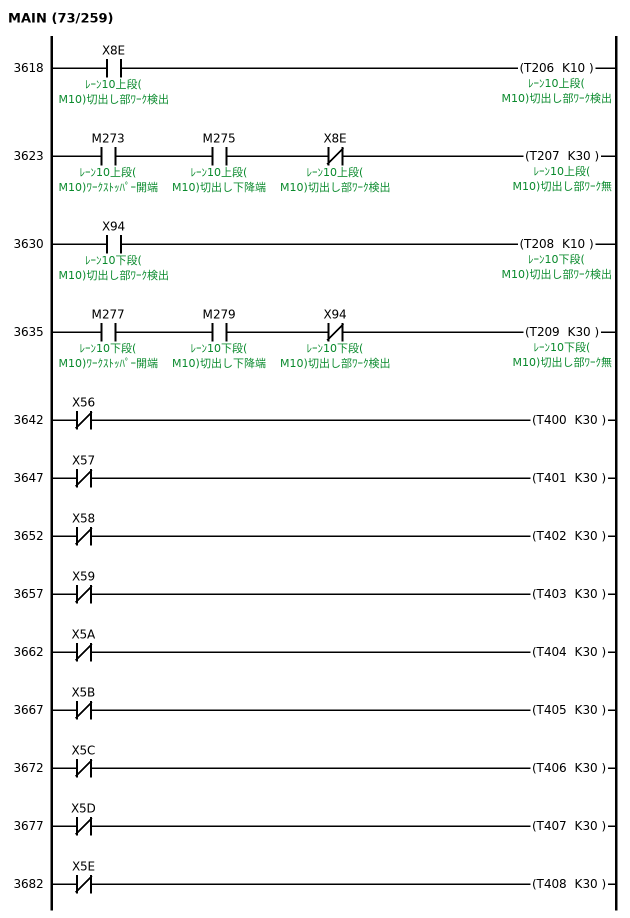
[picture p72: ladder of MAIN, rungs at steps 3618 to 3682]
3618  LD      X8E  ; ﾚｰﾝ10上段(M10)切出し部ﾜｰｸ検出
      OUT     T206 K10  ; ﾚｰﾝ10上段(M10)切出し部ﾜｰｸ検出
3623  LD      M273  ; ﾚｰﾝ10上段(M10)ﾜｰｸｽﾄｯﾊﾟｰ開端
      AND     M275  ; ﾚｰﾝ10上段(M10)切出し下降端
      ANI     X8E  ; ﾚｰﾝ10上段(M10)切出し部ﾜｰｸ検出
      OUT     T207 K30  ; ﾚｰﾝ10上段(M10)切出し部ﾜｰｸ無
3630  LD      X94  ; ﾚｰﾝ10下段(M10)切出し部ﾜｰｸ検出
      OUT     T208 K10  ; ﾚｰﾝ10下段(M10)切出し部ﾜｰｸ検出
3635  LD      M277  ; ﾚｰﾝ10下段(M10)ﾜｰｸｽﾄｯﾊﾟｰ開端
      AND     M279  ; ﾚｰﾝ10下段(M10)切出し下降端
      ANI     X94  ; ﾚｰﾝ10下段(M10)切出し部ﾜｰｸ検出
      OUT     T209 K30  ; ﾚｰﾝ10下段(M10)切出し部ﾜｰｸ無
3642  LDI     X56
      OUT     T400 K30
3647  LDI     X57
      OUT     T401 K30
3652  LDI     X58
      OUT     T402 K30
3657  LDI     X59
      OUT     T403 K30
3662  LDI     X5A
      OUT     T404 K30
3667  LDI     X5B
      OUT     T405 K30
3672  LDI     X5C
      OUT     T406 K30
3677  LDI     X5D
      OUT     T407 K30
3682  LDI     X5E
      OUT     T408 K30
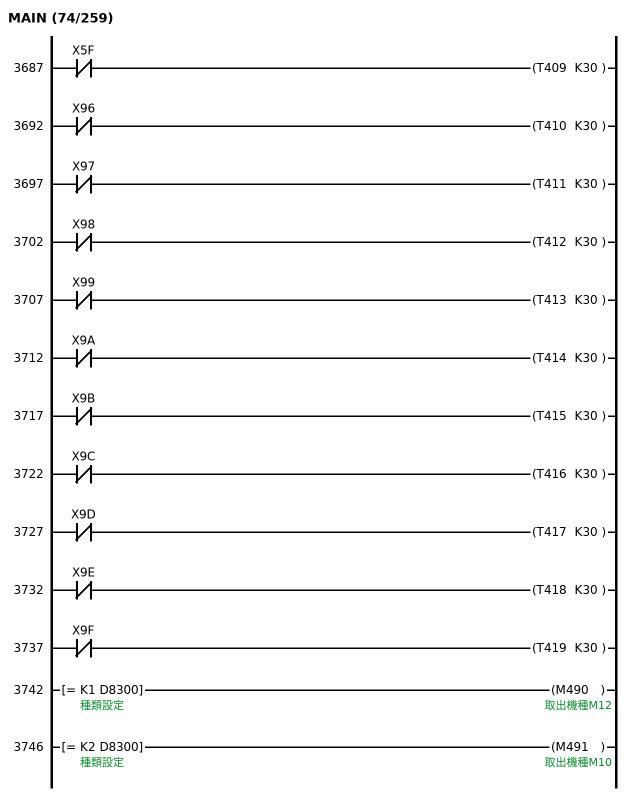
3687  LDI     X5F
      OUT     T409 K30
3692  LDI     X96
      OUT     T410 K30
3697  LDI     X97
      OUT     T411 K30
3702  LDI     X98
      OUT     T412 K30
3707  LDI     X99
      OUT     T413 K30
3712  LDI     X9A
      OUT     T414 K30
3717  LDI     X9B
      OUT     T415 K30
3722  LDI     X9C
      OUT     T416 K30
3727  LDI     X9D
      OUT     T417 K30
3732  LDI     X9E
      OUT     T418 K30
3737  LDI     X9F
      OUT     T419 K30
3742  LD=     K1 D8300  ; 種類設定
      OUT     M490  ; 取出機種M12
3746  LD=     K2 D8300  ; 種類設定
      OUT     M491  ; 取出機種M10
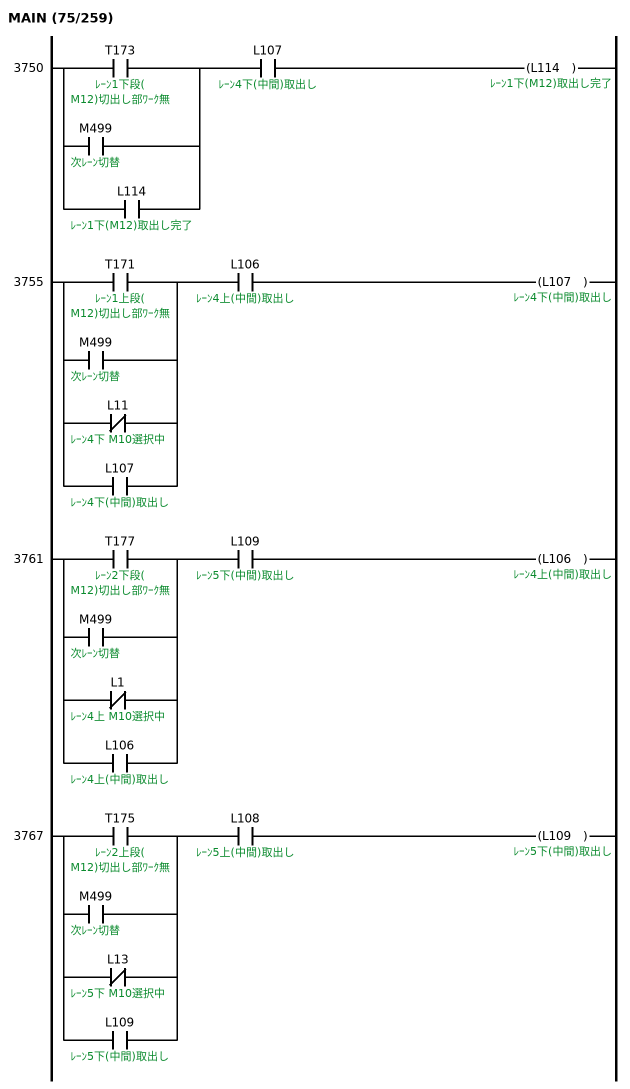
3750  LD      T173  ; ﾚｰﾝ1下段(M12)切出し部ﾜｰｸ無
      OR      M499  ; 次ﾚｰﾝ切替
      OR      L114  ; ﾚｰﾝ1下(M12)取出し完了
      AND     L107  ; ﾚｰﾝ4下(中間)取出し
      OUT     L114  ; ﾚｰﾝ1下(M12)取出し完了
3755  LD      T171  ; ﾚｰﾝ1上段(M12)切出し部ﾜｰｸ無
      OR      M499  ; 次ﾚｰﾝ切替
      ORI     L11  ; ﾚｰﾝ4下 M10選択中
      OR      L107  ; ﾚｰﾝ4下(中間)取出し
      AND     L106  ; ﾚｰﾝ4上(中間)取出し
      OUT     L107  ; ﾚｰﾝ4下(中間)取出し
3761  LD      T177  ; ﾚｰﾝ2下段(M12)切出し部ﾜｰｸ無
      OR      M499  ; 次ﾚｰﾝ切替
      ORI     L1  ; ﾚｰﾝ4上 M10選択中
      OR      L106  ; ﾚｰﾝ4上(中間)取出し
      AND     L109  ; ﾚｰﾝ5下(中間)取出し
      OUT     L106  ; ﾚｰﾝ4上(中間)取出し
3767  LD      T175  ; ﾚｰﾝ2上段(M12)切出し部ﾜｰｸ無
      OR      M499  ; 次ﾚｰﾝ切替
      ORI     L13  ; ﾚｰﾝ5下 M10選択中
      OR      L109  ; ﾚｰﾝ5下(中間)取出し
      AND     L108  ; ﾚｰﾝ5上(中間)取出し
      OUT     L109  ; ﾚｰﾝ5下(中間)取出し
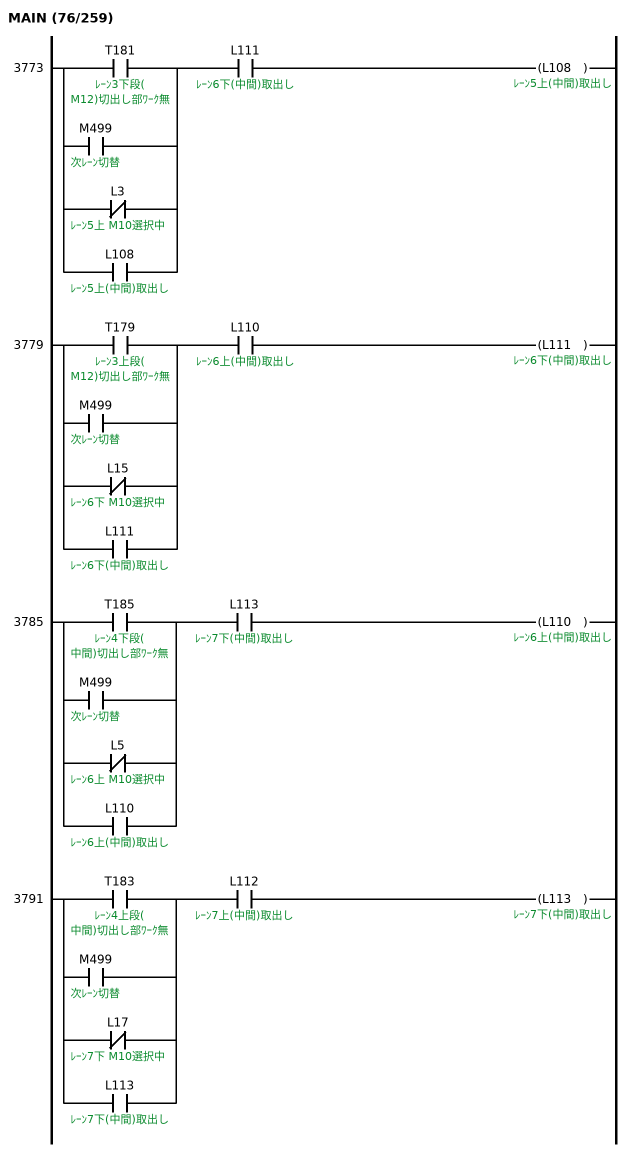
3773  LD      T181  ; ﾚｰﾝ3下段(M12)切出し部ﾜｰｸ無
      OR      M499  ; 次ﾚｰﾝ切替
      ORI     L3  ; ﾚｰﾝ5上 M10選択中
      OR      L108  ; ﾚｰﾝ5上(中間)取出し
      AND     L111  ; ﾚｰﾝ6下(中間)取出し
      OUT     L108  ; ﾚｰﾝ5上(中間)取出し
3779  LD      T179  ; ﾚｰﾝ3上段(M12)切出し部ﾜｰｸ無
      OR      M499  ; 次ﾚｰﾝ切替
      ORI     L15  ; ﾚｰﾝ6下 M10選択中
      OR      L111  ; ﾚｰﾝ6下(中間)取出し
      AND     L110  ; ﾚｰﾝ6上(中間)取出し
      OUT     L111  ; ﾚｰﾝ6下(中間)取出し
3785  LD      T185  ; ﾚｰﾝ4下段(中間)切出し部ﾜｰｸ無
      OR      M499  ; 次ﾚｰﾝ切替
      ORI     L5  ; ﾚｰﾝ6上 M10選択中
      OR      L110  ; ﾚｰﾝ6上(中間)取出し
      AND     L113  ; ﾚｰﾝ7下(中間)取出し
      OUT     L110  ; ﾚｰﾝ6上(中間)取出し
3791  LD      T183  ; ﾚｰﾝ4上段(中間)切出し部ﾜｰｸ無
      OR      M499  ; 次ﾚｰﾝ切替
      ORI     L17  ; ﾚｰﾝ7下 M10選択中
      OR      L113  ; ﾚｰﾝ7下(中間)取出し
      AND     L112  ; ﾚｰﾝ7上(中間)取出し
      OUT     L113  ; ﾚｰﾝ7下(中間)取出し
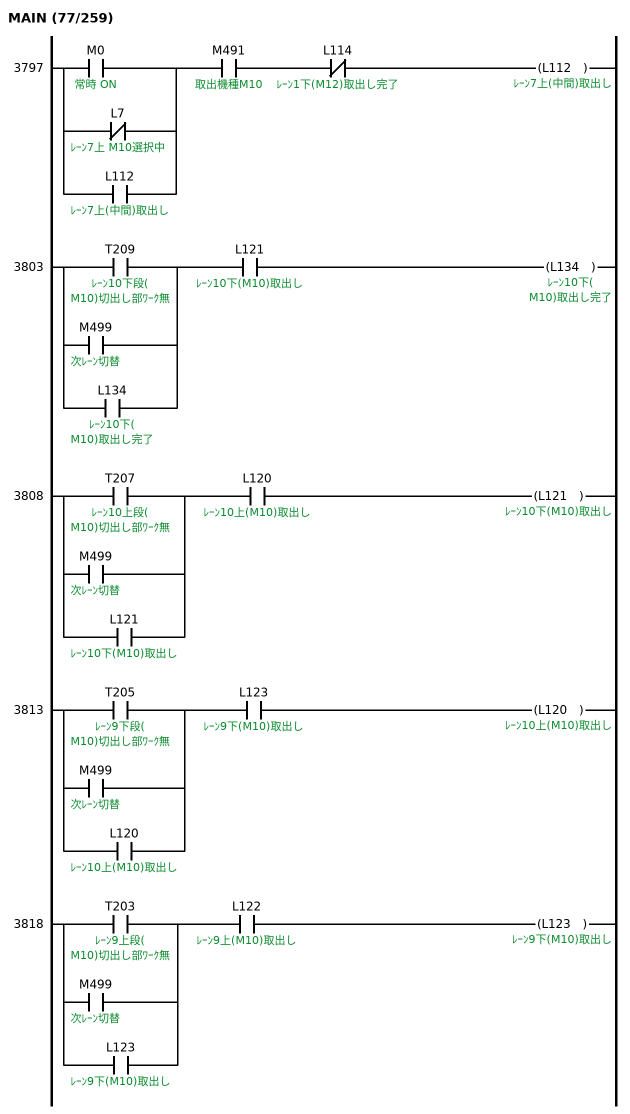
3797  LD      M0  ; 常時 ON
      ORI     L7  ; ﾚｰﾝ7上 M10選択中
      OR      L112  ; ﾚｰﾝ7上(中間)取出し
      AND     M491  ; 取出機種M10
      ANI     L114  ; ﾚｰﾝ1下(M12)取出し完了
      OUT     L112  ; ﾚｰﾝ7上(中間)取出し
3803  LD      T209  ; ﾚｰﾝ10下段(M10)切出し部ﾜｰｸ無
      OR      M499  ; 次ﾚｰﾝ切替
      OR      L134  ; ﾚｰﾝ10下(M10)取出し完了
      AND     L121  ; ﾚｰﾝ10下(M10)取出し
      OUT     L134  ; ﾚｰﾝ10下(M10)取出し完了
3808  LD      T207  ; ﾚｰﾝ10上段(M10)切出し部ﾜｰｸ無
      OR      M499  ; 次ﾚｰﾝ切替
      OR      L121  ; ﾚｰﾝ10下(M10)取出し
      AND     L120  ; ﾚｰﾝ10上(M10)取出し
      OUT     L121  ; ﾚｰﾝ10下(M10)取出し
3813  LD      T205  ; ﾚｰﾝ9下段(M10)切出し部ﾜｰｸ無
      OR      M499  ; 次ﾚｰﾝ切替
      OR      L120  ; ﾚｰﾝ10上(M10)取出し
      AND     L123  ; ﾚｰﾝ9下(M10)取出し
      OUT     L120  ; ﾚｰﾝ10上(M10)取出し
3818  LD      T203  ; ﾚｰﾝ9上段(M10)切出し部ﾜｰｸ無
      OR      M499  ; 次ﾚｰﾝ切替
      OR      L123  ; ﾚｰﾝ9下(M10)取出し
      AND     L122  ; ﾚｰﾝ9上(M10)取出し
      OUT     L123  ; ﾚｰﾝ9下(M10)取出し
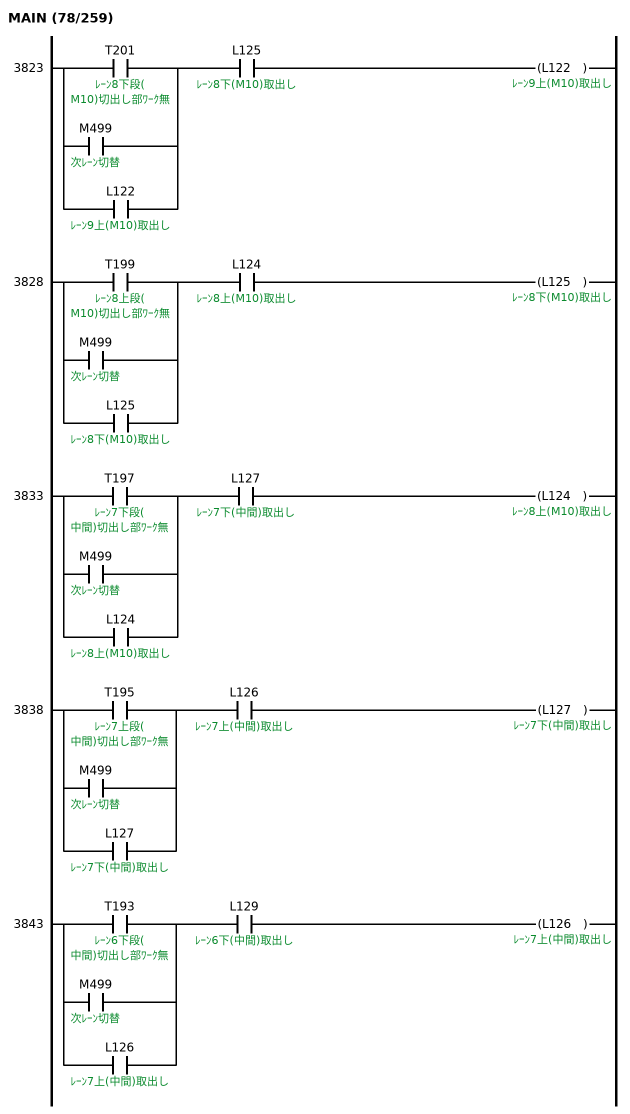
3823  LD      T201  ; ﾚｰﾝ8下段(M10)切出し部ﾜｰｸ無
      OR      M499  ; 次ﾚｰﾝ切替
      OR      L122  ; ﾚｰﾝ9上(M10)取出し
      AND     L125  ; ﾚｰﾝ8下(M10)取出し
      OUT     L122  ; ﾚｰﾝ9上(M10)取出し
3828  LD      T199  ; ﾚｰﾝ8上段(M10)切出し部ﾜｰｸ無
      OR      M499  ; 次ﾚｰﾝ切替
      OR      L125  ; ﾚｰﾝ8下(M10)取出し
      AND     L124  ; ﾚｰﾝ8上(M10)取出し
      OUT     L125  ; ﾚｰﾝ8下(M10)取出し
3833  LD      T197  ; ﾚｰﾝ7下段(中間)切出し部ﾜｰｸ無
      OR      M499  ; 次ﾚｰﾝ切替
      OR      L124  ; ﾚｰﾝ8上(M10)取出し
      AND     L127  ; ﾚｰﾝ7下(中間)取出し
      OUT     L124  ; ﾚｰﾝ8上(M10)取出し
3838  LD      T195  ; ﾚｰﾝ7上段(中間)切出し部ﾜｰｸ無
      OR      M499  ; 次ﾚｰﾝ切替
      OR      L127  ; ﾚｰﾝ7下(中間)取出し
      AND     L126  ; ﾚｰﾝ7上(中間)取出し
      OUT     L127  ; ﾚｰﾝ7下(中間)取出し
3843  LD      T193  ; ﾚｰﾝ6下段(中間)切出し部ﾜｰｸ無
      OR      M499  ; 次ﾚｰﾝ切替
      OR      L126  ; ﾚｰﾝ7上(中間)取出し
      AND     L129  ; ﾚｰﾝ6下(中間)取出し
      OUT     L126  ; ﾚｰﾝ7上(中間)取出し
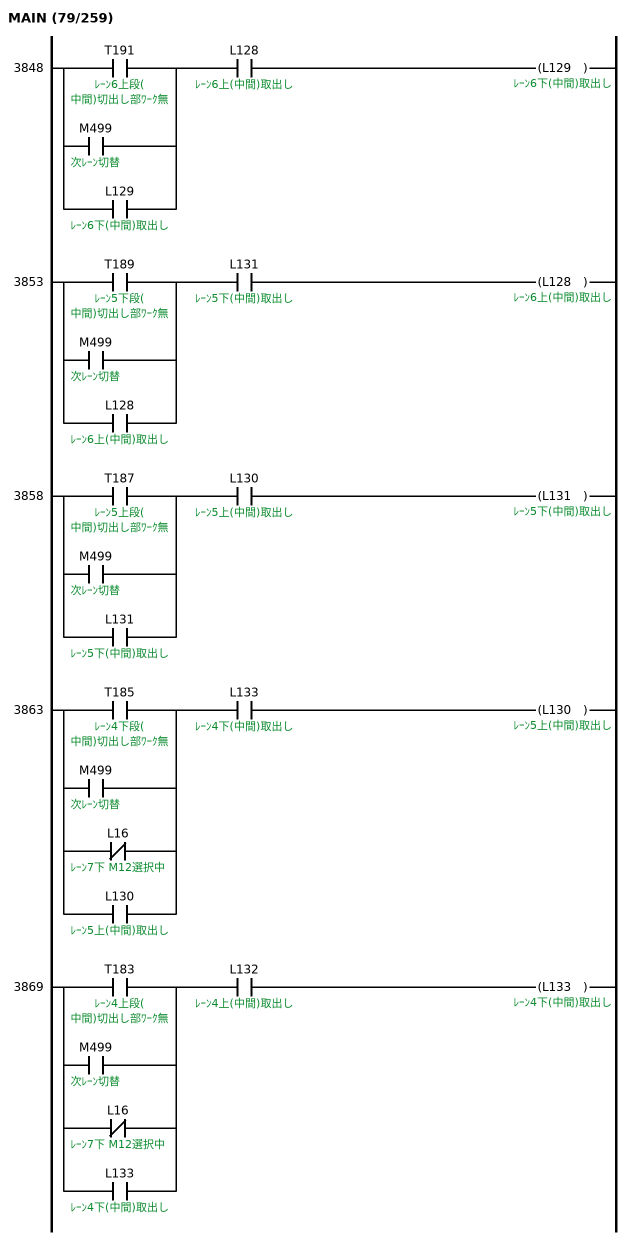
3848  LD      T191  ; ﾚｰﾝ6上段(中間)切出し部ﾜｰｸ無
      OR      M499  ; 次ﾚｰﾝ切替
      OR      L129  ; ﾚｰﾝ6下(中間)取出し
      AND     L128  ; ﾚｰﾝ6上(中間)取出し
      OUT     L129  ; ﾚｰﾝ6下(中間)取出し
3853  LD      T189  ; ﾚｰﾝ5下段(中間)切出し部ﾜｰｸ無
      OR      M499  ; 次ﾚｰﾝ切替
      OR      L128  ; ﾚｰﾝ6上(中間)取出し
      AND     L131  ; ﾚｰﾝ5下(中間)取出し
      OUT     L128  ; ﾚｰﾝ6上(中間)取出し
3858  LD      T187  ; ﾚｰﾝ5上段(中間)切出し部ﾜｰｸ無
      OR      M499  ; 次ﾚｰﾝ切替
      OR      L131  ; ﾚｰﾝ5下(中間)取出し
      AND     L130  ; ﾚｰﾝ5上(中間)取出し
      OUT     L131  ; ﾚｰﾝ5下(中間)取出し
3863  LD      T185  ; ﾚｰﾝ4下段(中間)切出し部ﾜｰｸ無
      OR      M499  ; 次ﾚｰﾝ切替
      ORI     L16  ; ﾚｰﾝ7下 M12選択中
      OR      L130  ; ﾚｰﾝ5上(中間)取出し
      AND     L133  ; ﾚｰﾝ4下(中間)取出し
      OUT     L130  ; ﾚｰﾝ5上(中間)取出し
3869  LD      T183  ; ﾚｰﾝ4上段(中間)切出し部ﾜｰｸ無
      OR      M499  ; 次ﾚｰﾝ切替
      ORI     L16  ; ﾚｰﾝ7下 M12選択中
      OR      L133  ; ﾚｰﾝ4下(中間)取出し
      AND     L132  ; ﾚｰﾝ4上(中間)取出し
      OUT     L133  ; ﾚｰﾝ4下(中間)取出し
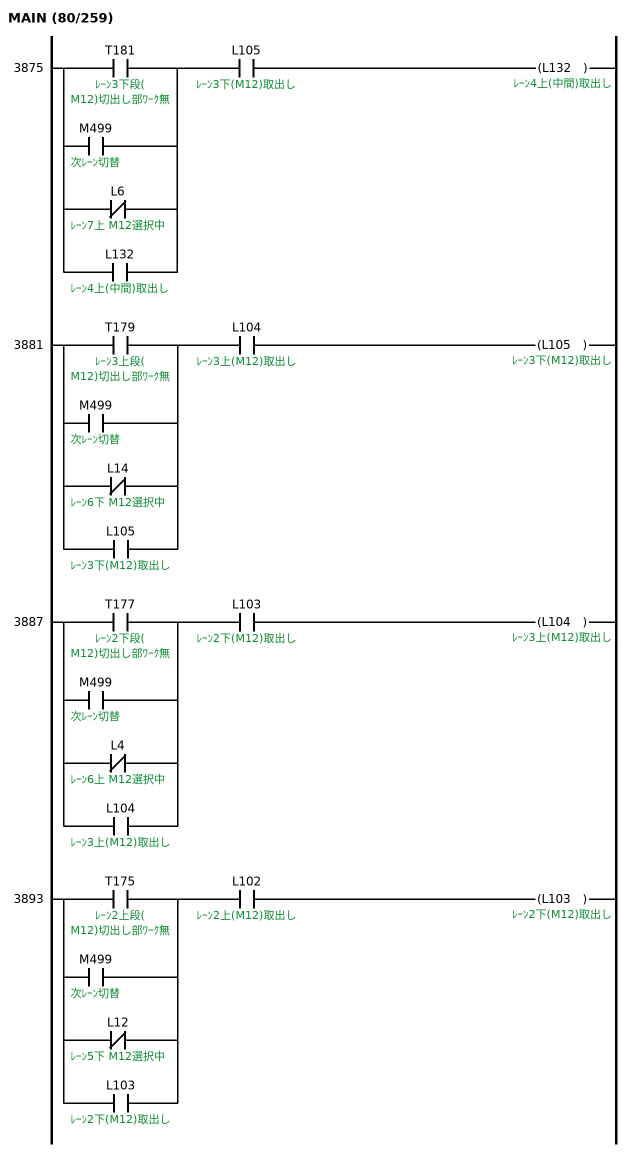
3875  LD      T181  ; ﾚｰﾝ3下段(M12)切出し部ﾜｰｸ無
      OR      M499  ; 次ﾚｰﾝ切替
      ORI     L6  ; ﾚｰﾝ7上 M12選択中
      OR      L132  ; ﾚｰﾝ4上(中間)取出し
      AND     L105  ; ﾚｰﾝ3下(M12)取出し
      OUT     L132  ; ﾚｰﾝ4上(中間)取出し
3881  LD      T179  ; ﾚｰﾝ3上段(M12)切出し部ﾜｰｸ無
      OR      M499  ; 次ﾚｰﾝ切替
      ORI     L14  ; ﾚｰﾝ6下 M12選択中
      OR      L105  ; ﾚｰﾝ3下(M12)取出し
      AND     L104  ; ﾚｰﾝ3上(M12)取出し
      OUT     L105  ; ﾚｰﾝ3下(M12)取出し
3887  LD      T177  ; ﾚｰﾝ2下段(M12)切出し部ﾜｰｸ無
      OR      M499  ; 次ﾚｰﾝ切替
      ORI     L4  ; ﾚｰﾝ6上 M12選択中
      OR      L104  ; ﾚｰﾝ3上(M12)取出し
      AND     L103  ; ﾚｰﾝ2下(M12)取出し
      OUT     L104  ; ﾚｰﾝ3上(M12)取出し
3893  LD      T175  ; ﾚｰﾝ2上段(M12)切出し部ﾜｰｸ無
      OR      M499  ; 次ﾚｰﾝ切替
      ORI     L12  ; ﾚｰﾝ5下 M12選択中
      OR      L103  ; ﾚｰﾝ2下(M12)取出し
      AND     L102  ; ﾚｰﾝ2上(M12)取出し
      OUT     L103  ; ﾚｰﾝ2下(M12)取出し
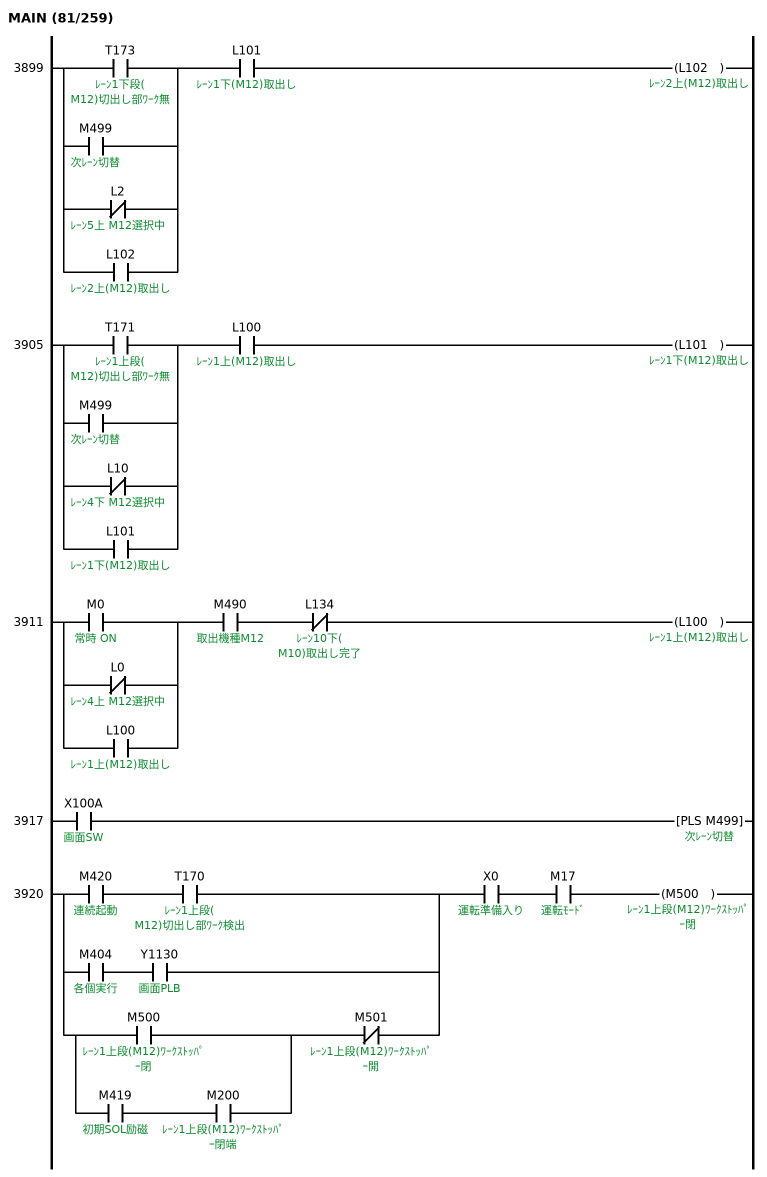
3899  LD      T173  ; ﾚｰﾝ1下段(M12)切出し部ﾜｰｸ無
      OR      M499  ; 次ﾚｰﾝ切替
      ORI     L2  ; ﾚｰﾝ5上 M12選択中
      OR      L102  ; ﾚｰﾝ2上(M12)取出し
      AND     L101  ; ﾚｰﾝ1下(M12)取出し
      OUT     L102  ; ﾚｰﾝ2上(M12)取出し
3905  LD      T171  ; ﾚｰﾝ1上段(M12)切出し部ﾜｰｸ無
      OR      M499  ; 次ﾚｰﾝ切替
      ORI     L10  ; ﾚｰﾝ4下 M12選択中
      OR      L101  ; ﾚｰﾝ1下(M12)取出し
      AND     L100  ; ﾚｰﾝ1上(M12)取出し
      OUT     L101  ; ﾚｰﾝ1下(M12)取出し
3911  LD      M0  ; 常時 ON
      ORI     L0  ; ﾚｰﾝ4上 M12選択中
      OR      L100  ; ﾚｰﾝ1上(M12)取出し
      AND     M490  ; 取出機種M12
      ANI     L134  ; ﾚｰﾝ10下(M10)取出し完了
      OUT     L100  ; ﾚｰﾝ1上(M12)取出し
3917  LD      X100A  ; 画面SW
      PLS     M499  ; 次ﾚｰﾝ切替
3920  LD      M420  ; 連続起動
      AND     T170  ; ﾚｰﾝ1上段(M12)切出し部ﾜｰｸ検出
      LD      M404  ; 各個実行
      AND     Y1130  ; 画面PLB
      ORB
      LD      M500  ; ﾚｰﾝ1上段(M12)ﾜｰｸｽﾄｯﾊﾟｰ閉
      LD      M419  ; 初期SOL励磁
      AND     M200  ; ﾚｰﾝ1上段(M12)ﾜｰｸｽﾄｯﾊﾟｰ閉端
      ORB
      ANI     M501  ; ﾚｰﾝ1上段(M12)ﾜｰｸｽﾄｯﾊﾟｰ開
      ORB
      AND     X0  ; 運転準備入り
      AND     M17  ; 運転ﾓｰﾄﾞ
      OUT     M500  ; ﾚｰﾝ1上段(M12)ﾜｰｸｽﾄｯﾊﾟｰ閉
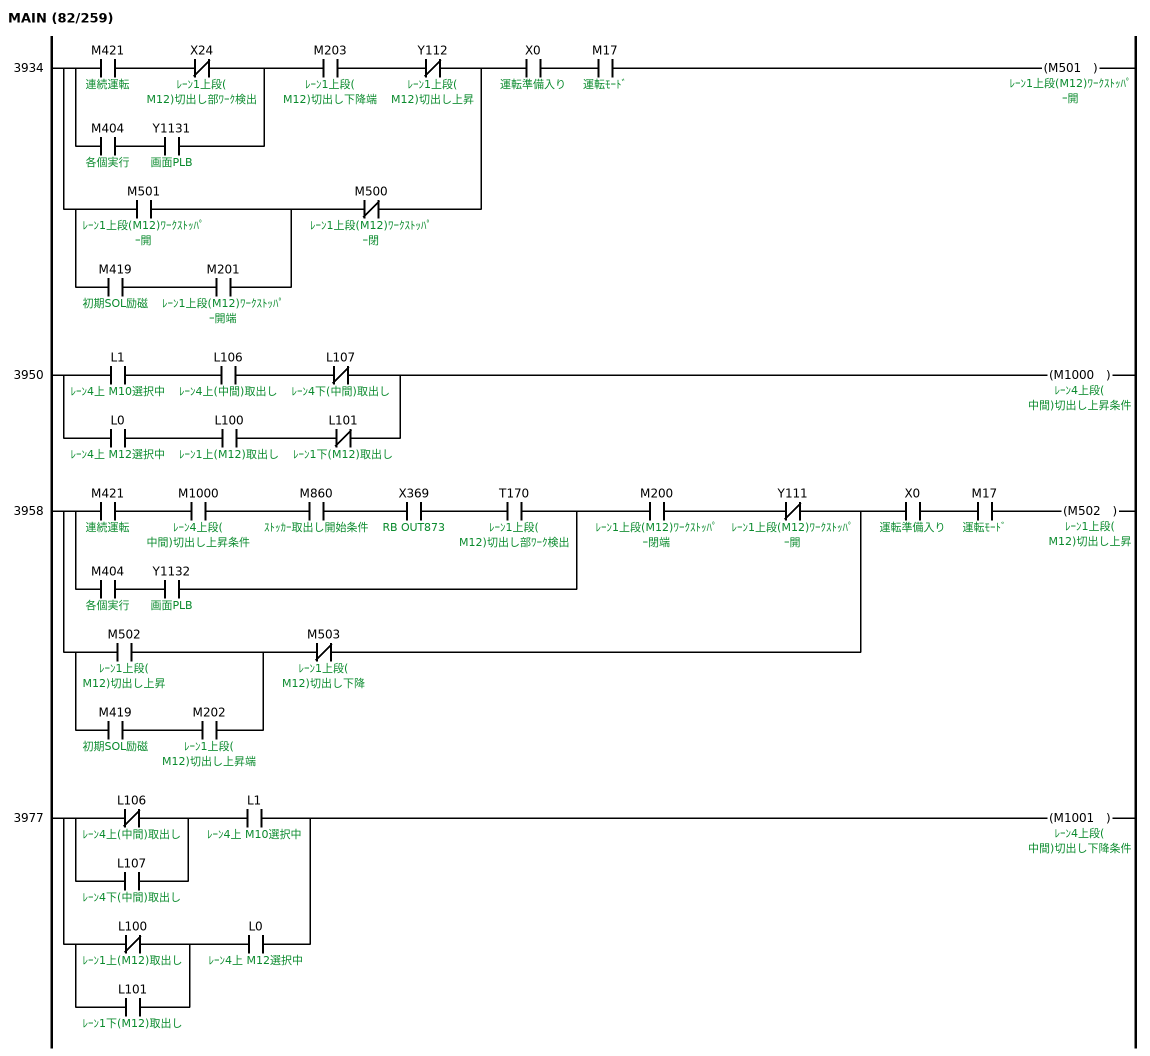
3934  LD      M421  ; 連続運転
      ANI     X24  ; ﾚｰﾝ1上段(M12)切出し部ﾜｰｸ検出
      LD      M404  ; 各個実行
      AND     Y1131  ; 画面PLB
      ORB
      AND     M203  ; ﾚｰﾝ1上段(M12)切出し下降端
      ANI     Y112  ; ﾚｰﾝ1上段(M12)切出し上昇
      LD      M501  ; ﾚｰﾝ1上段(M12)ﾜｰｸｽﾄｯﾊﾟｰ開
      LD      M419  ; 初期SOL励磁
      AND     M201  ; ﾚｰﾝ1上段(M12)ﾜｰｸｽﾄｯﾊﾟｰ開端
      ORB
      ANI     M500  ; ﾚｰﾝ1上段(M12)ﾜｰｸｽﾄｯﾊﾟｰ閉
      ORB
      AND     X0  ; 運転準備入り
      AND     M17  ; 運転ﾓｰﾄﾞ
      OUT     M501  ; ﾚｰﾝ1上段(M12)ﾜｰｸｽﾄｯﾊﾟｰ開
3950  LD      L1  ; ﾚｰﾝ4上 M10選択中
      AND     L106  ; ﾚｰﾝ4上(中間)取出し
      ANI     L107  ; ﾚｰﾝ4下(中間)取出し
      LD      L0  ; ﾚｰﾝ4上 M12選択中
      AND     L100  ; ﾚｰﾝ1上(M12)取出し
      ANI     L101  ; ﾚｰﾝ1下(M12)取出し
      ORB
      OUT     M1000  ; ﾚｰﾝ4上段(中間)切出し上昇条件
3958  LD      M421  ; 連続運転
      AND     M1000  ; ﾚｰﾝ4上段(中間)切出し上昇条件
      AND     M860  ; ｽﾄｯｶｰ取出し開始条件
      AND     X369  ; RB OUT873
      AND     T170  ; ﾚｰﾝ1上段(M12)切出し部ﾜｰｸ検出
      LD      M404  ; 各個実行
      AND     Y1132  ; 画面PLB
      ORB
      AND     M200  ; ﾚｰﾝ1上段(M12)ﾜｰｸｽﾄｯﾊﾟｰ閉端
      ANI     Y111  ; ﾚｰﾝ1上段(M12)ﾜｰｸｽﾄｯﾊﾟｰ開
      LD      M502  ; ﾚｰﾝ1上段(M12)切出し上昇
      LD      M419  ; 初期SOL励磁
      AND     M202  ; ﾚｰﾝ1上段(M12)切出し上昇端
      ORB
      ANI     M503  ; ﾚｰﾝ1上段(M12)切出し下降
      ORB
      AND     X0  ; 運転準備入り
      AND     M17  ; 運転ﾓｰﾄﾞ
      OUT     M502  ; ﾚｰﾝ1上段(M12)切出し上昇
3977  LDI     L106  ; ﾚｰﾝ4上(中間)取出し
      OR      L107  ; ﾚｰﾝ4下(中間)取出し
      AND     L1  ; ﾚｰﾝ4上 M10選択中
      LDI     L100  ; ﾚｰﾝ1上(M12)取出し
      OR      L101  ; ﾚｰﾝ1下(M12)取出し
      AND     L0  ; ﾚｰﾝ4上 M12選択中
      ORB
      OUT     M1001  ; ﾚｰﾝ4上段(中間)切出し下降条件
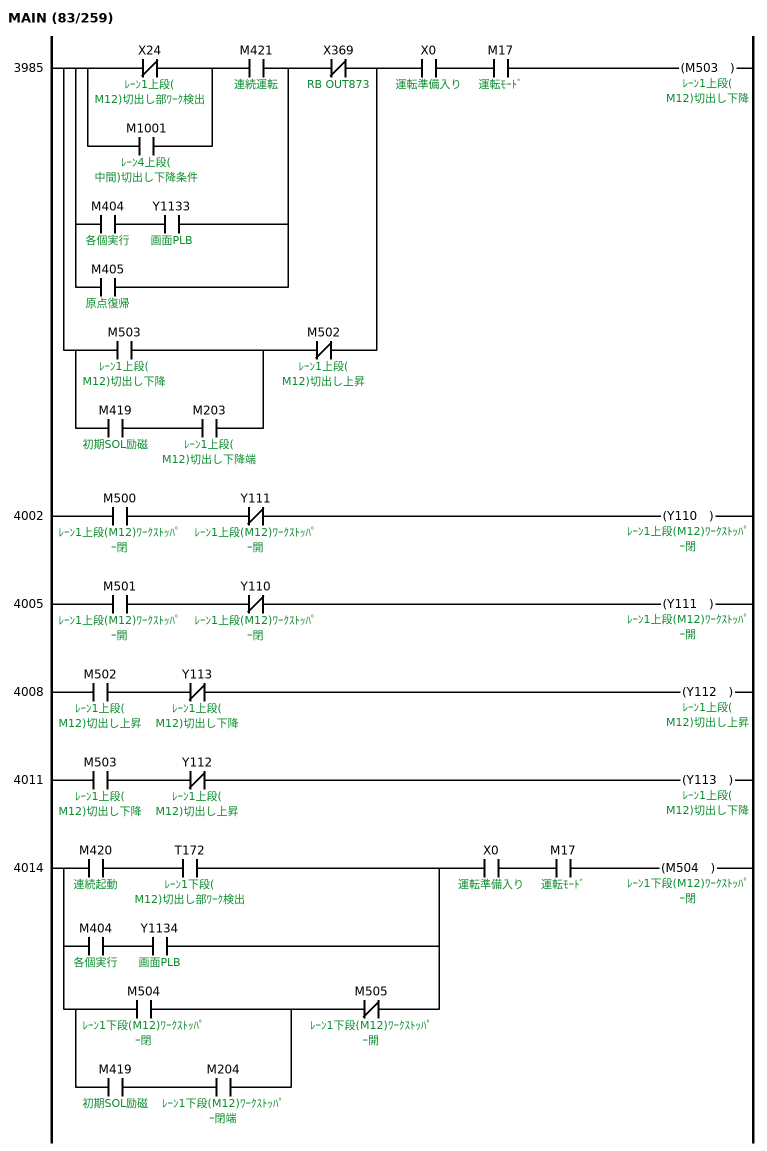
3985  LDI     X24  ; ﾚｰﾝ1上段(M12)切出し部ﾜｰｸ検出
      OR      M1001  ; ﾚｰﾝ4上段(中間)切出し下降条件
      AND     M421  ; 連続運転
      LD      M404  ; 各個実行
      AND     Y1133  ; 画面PLB
      ORB
      OR      M405  ; 原点復帰
      ANI     X369  ; RB OUT873
      LD      M503  ; ﾚｰﾝ1上段(M12)切出し下降
      LD      M419  ; 初期SOL励磁
      AND     M203  ; ﾚｰﾝ1上段(M12)切出し下降端
      ORB
      ANI     M502  ; ﾚｰﾝ1上段(M12)切出し上昇
      ORB
      AND     X0  ; 運転準備入り
      AND     M17  ; 運転ﾓｰﾄﾞ
      OUT     M503  ; ﾚｰﾝ1上段(M12)切出し下降
4002  LD      M500  ; ﾚｰﾝ1上段(M12)ﾜｰｸｽﾄｯﾊﾟｰ閉
      ANI     Y111  ; ﾚｰﾝ1上段(M12)ﾜｰｸｽﾄｯﾊﾟｰ開
      OUT     Y110  ; ﾚｰﾝ1上段(M12)ﾜｰｸｽﾄｯﾊﾟｰ閉
4005  LD      M501  ; ﾚｰﾝ1上段(M12)ﾜｰｸｽﾄｯﾊﾟｰ開
      ANI     Y110  ; ﾚｰﾝ1上段(M12)ﾜｰｸｽﾄｯﾊﾟｰ閉
      OUT     Y111  ; ﾚｰﾝ1上段(M12)ﾜｰｸｽﾄｯﾊﾟｰ開
4008  LD      M502  ; ﾚｰﾝ1上段(M12)切出し上昇
      ANI     Y113  ; ﾚｰﾝ1上段(M12)切出し下降
      OUT     Y112  ; ﾚｰﾝ1上段(M12)切出し上昇
4011  LD      M503  ; ﾚｰﾝ1上段(M12)切出し下降
      ANI     Y112  ; ﾚｰﾝ1上段(M12)切出し上昇
      OUT     Y113  ; ﾚｰﾝ1上段(M12)切出し下降
4014  LD      M420  ; 連続起動
      AND     T172  ; ﾚｰﾝ1下段(M12)切出し部ﾜｰｸ検出
      LD      M404  ; 各個実行
      AND     Y1134  ; 画面PLB
      ORB
      LD      M504  ; ﾚｰﾝ1下段(M12)ﾜｰｸｽﾄｯﾊﾟｰ閉
      LD      M419  ; 初期SOL励磁
      AND     M204  ; ﾚｰﾝ1下段(M12)ﾜｰｸｽﾄｯﾊﾟｰ閉端
      ORB
      ANI     M505  ; ﾚｰﾝ1下段(M12)ﾜｰｸｽﾄｯﾊﾟｰ開
      ORB
      AND     X0  ; 運転準備入り
      AND     M17  ; 運転ﾓｰﾄﾞ
      OUT     M504  ; ﾚｰﾝ1下段(M12)ﾜｰｸｽﾄｯﾊﾟｰ閉
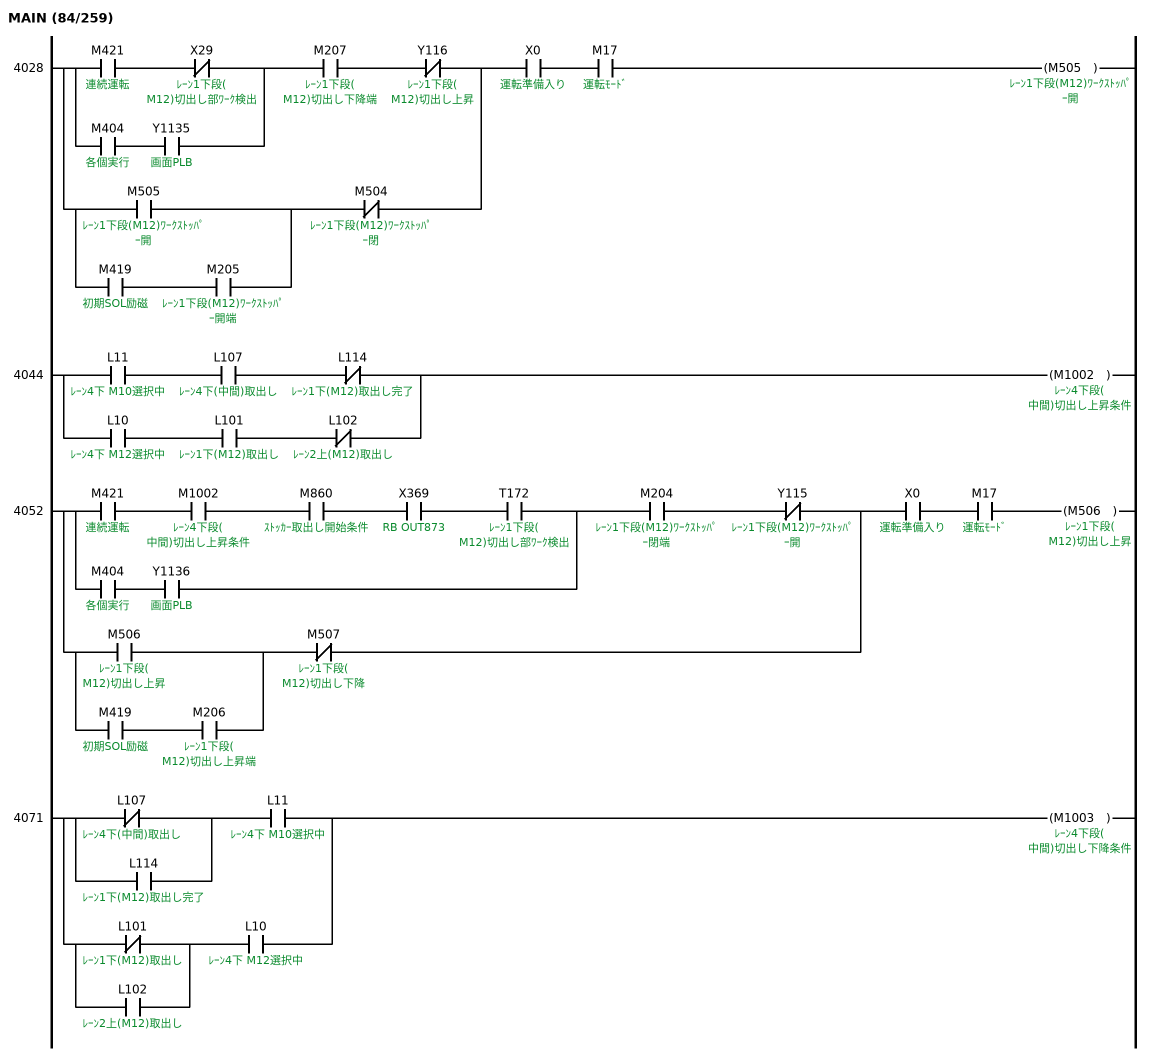
4028  LD      M421  ; 連続運転
      ANI     X29  ; ﾚｰﾝ1下段(M12)切出し部ﾜｰｸ検出
      LD      M404  ; 各個実行
      AND     Y1135  ; 画面PLB
      ORB
      AND     M207  ; ﾚｰﾝ1下段(M12)切出し下降端
      ANI     Y116  ; ﾚｰﾝ1下段(M12)切出し上昇
      LD      M505  ; ﾚｰﾝ1下段(M12)ﾜｰｸｽﾄｯﾊﾟｰ開
      LD      M419  ; 初期SOL励磁
      AND     M205  ; ﾚｰﾝ1下段(M12)ﾜｰｸｽﾄｯﾊﾟｰ開端
      ORB
      ANI     M504  ; ﾚｰﾝ1下段(M12)ﾜｰｸｽﾄｯﾊﾟｰ閉
      ORB
      AND     X0  ; 運転準備入り
      AND     M17  ; 運転ﾓｰﾄﾞ
      OUT     M505  ; ﾚｰﾝ1下段(M12)ﾜｰｸｽﾄｯﾊﾟｰ開
4044  LD      L11  ; ﾚｰﾝ4下 M10選択中
      AND     L107  ; ﾚｰﾝ4下(中間)取出し
      ANI     L114  ; ﾚｰﾝ1下(M12)取出し完了
      LD      L10  ; ﾚｰﾝ4下 M12選択中
      AND     L101  ; ﾚｰﾝ1下(M12)取出し
      ANI     L102  ; ﾚｰﾝ2上(M12)取出し
      ORB
      OUT     M1002  ; ﾚｰﾝ4下段(中間)切出し上昇条件
4052  LD      M421  ; 連続運転
      AND     M1002  ; ﾚｰﾝ4下段(中間)切出し上昇条件
      AND     M860  ; ｽﾄｯｶｰ取出し開始条件
      AND     X369  ; RB OUT873
      AND     T172  ; ﾚｰﾝ1下段(M12)切出し部ﾜｰｸ検出
      LD      M404  ; 各個実行
      AND     Y1136  ; 画面PLB
      ORB
      AND     M204  ; ﾚｰﾝ1下段(M12)ﾜｰｸｽﾄｯﾊﾟｰ閉端
      ANI     Y115  ; ﾚｰﾝ1下段(M12)ﾜｰｸｽﾄｯﾊﾟｰ開
      LD      M506  ; ﾚｰﾝ1下段(M12)切出し上昇
      LD      M419  ; 初期SOL励磁
      AND     M206  ; ﾚｰﾝ1下段(M12)切出し上昇端
      ORB
      ANI     M507  ; ﾚｰﾝ1下段(M12)切出し下降
      ORB
      AND     X0  ; 運転準備入り
      AND     M17  ; 運転ﾓｰﾄﾞ
      OUT     M506  ; ﾚｰﾝ1下段(M12)切出し上昇
4071  LDI     L107  ; ﾚｰﾝ4下(中間)取出し
      OR      L114  ; ﾚｰﾝ1下(M12)取出し完了
      AND     L11  ; ﾚｰﾝ4下 M10選択中
      LDI     L101  ; ﾚｰﾝ1下(M12)取出し
      OR      L102  ; ﾚｰﾝ2上(M12)取出し
      AND     L10  ; ﾚｰﾝ4下 M12選択中
      ORB
      OUT     M1003  ; ﾚｰﾝ4下段(中間)切出し下降条件
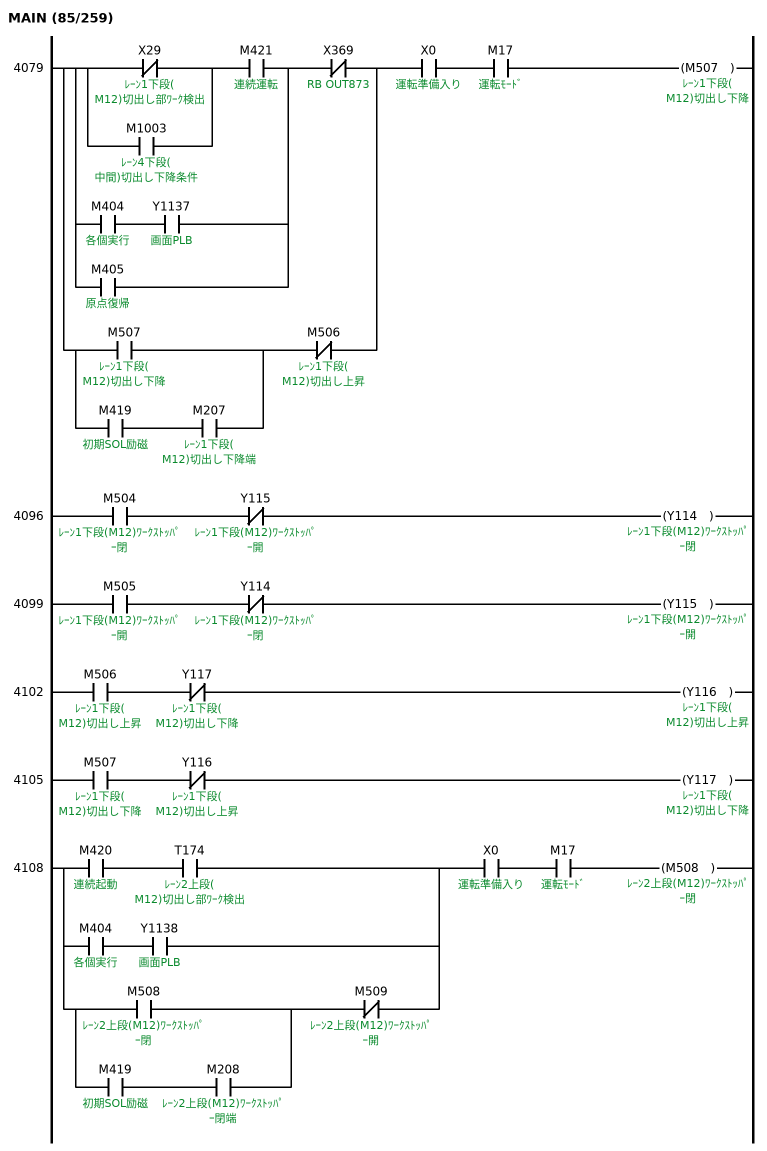
4079  LDI     X29  ; ﾚｰﾝ1下段(M12)切出し部ﾜｰｸ検出
      OR      M1003  ; ﾚｰﾝ4下段(中間)切出し下降条件
      AND     M421  ; 連続運転
      LD      M404  ; 各個実行
      AND     Y1137  ; 画面PLB
      ORB
      OR      M405  ; 原点復帰
      ANI     X369  ; RB OUT873
      LD      M507  ; ﾚｰﾝ1下段(M12)切出し下降
      LD      M419  ; 初期SOL励磁
      AND     M207  ; ﾚｰﾝ1下段(M12)切出し下降端
      ORB
      ANI     M506  ; ﾚｰﾝ1下段(M12)切出し上昇
      ORB
      AND     X0  ; 運転準備入り
      AND     M17  ; 運転ﾓｰﾄﾞ
      OUT     M507  ; ﾚｰﾝ1下段(M12)切出し下降
4096  LD      M504  ; ﾚｰﾝ1下段(M12)ﾜｰｸｽﾄｯﾊﾟｰ閉
      ANI     Y115  ; ﾚｰﾝ1下段(M12)ﾜｰｸｽﾄｯﾊﾟｰ開
      OUT     Y114  ; ﾚｰﾝ1下段(M12)ﾜｰｸｽﾄｯﾊﾟｰ閉
4099  LD      M505  ; ﾚｰﾝ1下段(M12)ﾜｰｸｽﾄｯﾊﾟｰ開
      ANI     Y114  ; ﾚｰﾝ1下段(M12)ﾜｰｸｽﾄｯﾊﾟｰ閉
      OUT     Y115  ; ﾚｰﾝ1下段(M12)ﾜｰｸｽﾄｯﾊﾟｰ開
4102  LD      M506  ; ﾚｰﾝ1下段(M12)切出し上昇
      ANI     Y117  ; ﾚｰﾝ1下段(M12)切出し下降
      OUT     Y116  ; ﾚｰﾝ1下段(M12)切出し上昇
4105  LD      M507  ; ﾚｰﾝ1下段(M12)切出し下降
      ANI     Y116  ; ﾚｰﾝ1下段(M12)切出し上昇
      OUT     Y117  ; ﾚｰﾝ1下段(M12)切出し下降
4108  LD      M420  ; 連続起動
      AND     T174  ; ﾚｰﾝ2上段(M12)切出し部ﾜｰｸ検出
      LD      M404  ; 各個実行
      AND     Y1138  ; 画面PLB
      ORB
      LD      M508  ; ﾚｰﾝ2上段(M12)ﾜｰｸｽﾄｯﾊﾟｰ閉
      LD      M419  ; 初期SOL励磁
      AND     M208  ; ﾚｰﾝ2上段(M12)ﾜｰｸｽﾄｯﾊﾟｰ閉端
      ORB
      ANI     M509  ; ﾚｰﾝ2上段(M12)ﾜｰｸｽﾄｯﾊﾟｰ開
      ORB
      AND     X0  ; 運転準備入り
      AND     M17  ; 運転ﾓｰﾄﾞ
      OUT     M508  ; ﾚｰﾝ2上段(M12)ﾜｰｸｽﾄｯﾊﾟｰ閉
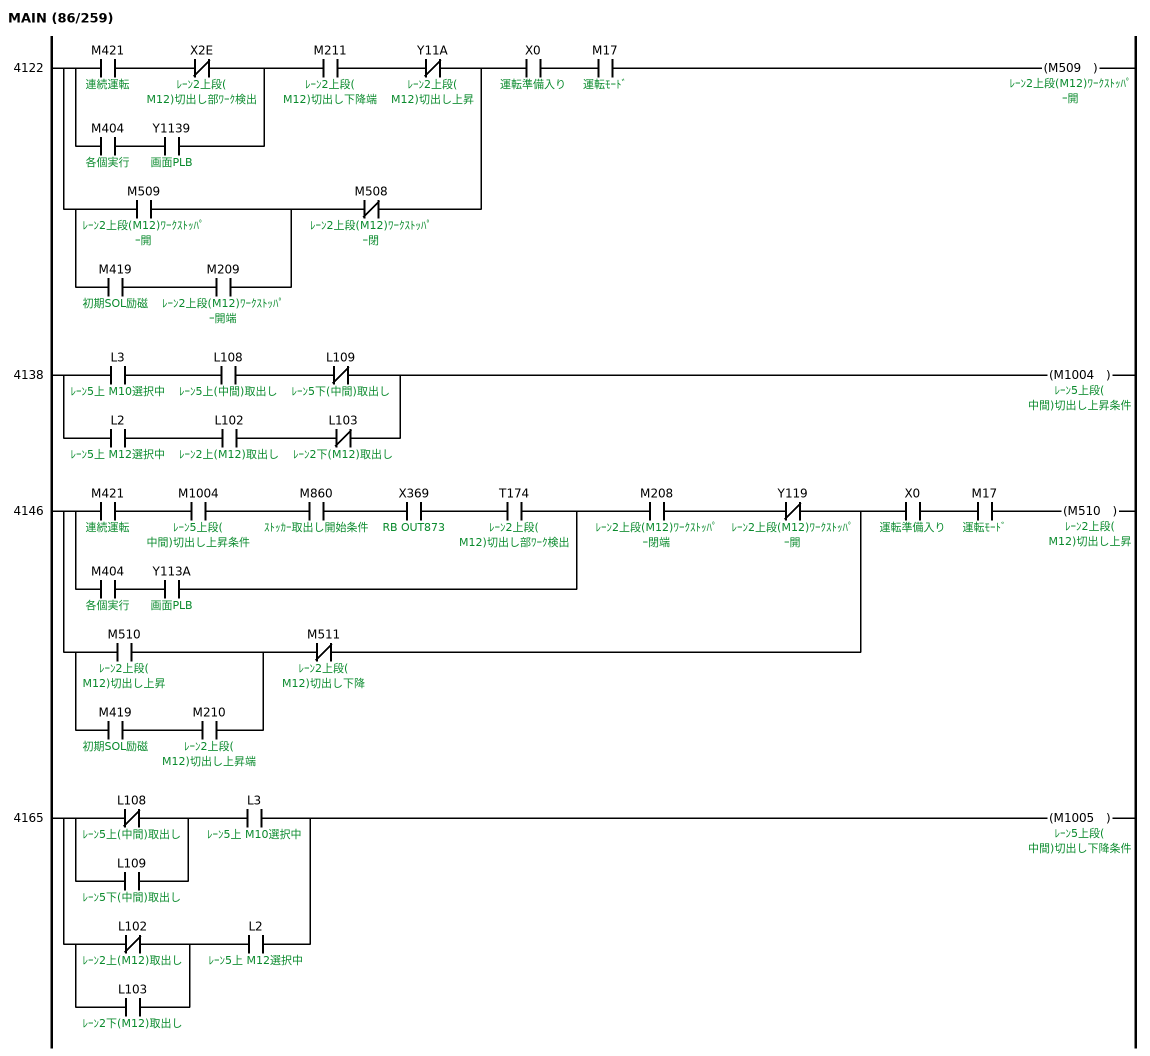
4122  LD      M421  ; 連続運転
      ANI     X2E  ; ﾚｰﾝ2上段(M12)切出し部ﾜｰｸ検出
      LD      M404  ; 各個実行
      AND     Y1139  ; 画面PLB
      ORB
      AND     M211  ; ﾚｰﾝ2上段(M12)切出し下降端
      ANI     Y11A  ; ﾚｰﾝ2上段(M12)切出し上昇
      LD      M509  ; ﾚｰﾝ2上段(M12)ﾜｰｸｽﾄｯﾊﾟｰ開
      LD      M419  ; 初期SOL励磁
      AND     M209  ; ﾚｰﾝ2上段(M12)ﾜｰｸｽﾄｯﾊﾟｰ開端
      ORB
      ANI     M508  ; ﾚｰﾝ2上段(M12)ﾜｰｸｽﾄｯﾊﾟｰ閉
      ORB
      AND     X0  ; 運転準備入り
      AND     M17  ; 運転ﾓｰﾄﾞ
      OUT     M509  ; ﾚｰﾝ2上段(M12)ﾜｰｸｽﾄｯﾊﾟｰ開
4138  LD      L3  ; ﾚｰﾝ5上 M10選択中
      AND     L108  ; ﾚｰﾝ5上(中間)取出し
      ANI     L109  ; ﾚｰﾝ5下(中間)取出し
      LD      L2  ; ﾚｰﾝ5上 M12選択中
      AND     L102  ; ﾚｰﾝ2上(M12)取出し
      ANI     L103  ; ﾚｰﾝ2下(M12)取出し
      ORB
      OUT     M1004  ; ﾚｰﾝ5上段(中間)切出し上昇条件
4146  LD      M421  ; 連続運転
      AND     M1004  ; ﾚｰﾝ5上段(中間)切出し上昇条件
      AND     M860  ; ｽﾄｯｶｰ取出し開始条件
      AND     X369  ; RB OUT873
      AND     T174  ; ﾚｰﾝ2上段(M12)切出し部ﾜｰｸ検出
      LD      M404  ; 各個実行
      AND     Y113A  ; 画面PLB
      ORB
      AND     M208  ; ﾚｰﾝ2上段(M12)ﾜｰｸｽﾄｯﾊﾟｰ閉端
      ANI     Y119  ; ﾚｰﾝ2上段(M12)ﾜｰｸｽﾄｯﾊﾟｰ開
      LD      M510  ; ﾚｰﾝ2上段(M12)切出し上昇
      LD      M419  ; 初期SOL励磁
      AND     M210  ; ﾚｰﾝ2上段(M12)切出し上昇端
      ORB
      ANI     M511  ; ﾚｰﾝ2上段(M12)切出し下降
      ORB
      AND     X0  ; 運転準備入り
      AND     M17  ; 運転ﾓｰﾄﾞ
      OUT     M510  ; ﾚｰﾝ2上段(M12)切出し上昇
4165  LDI     L108  ; ﾚｰﾝ5上(中間)取出し
      OR      L109  ; ﾚｰﾝ5下(中間)取出し
      AND     L3  ; ﾚｰﾝ5上 M10選択中
      LDI     L102  ; ﾚｰﾝ2上(M12)取出し
      OR      L103  ; ﾚｰﾝ2下(M12)取出し
      AND     L2  ; ﾚｰﾝ5上 M12選択中
      ORB
      OUT     M1005  ; ﾚｰﾝ5上段(中間)切出し下降条件
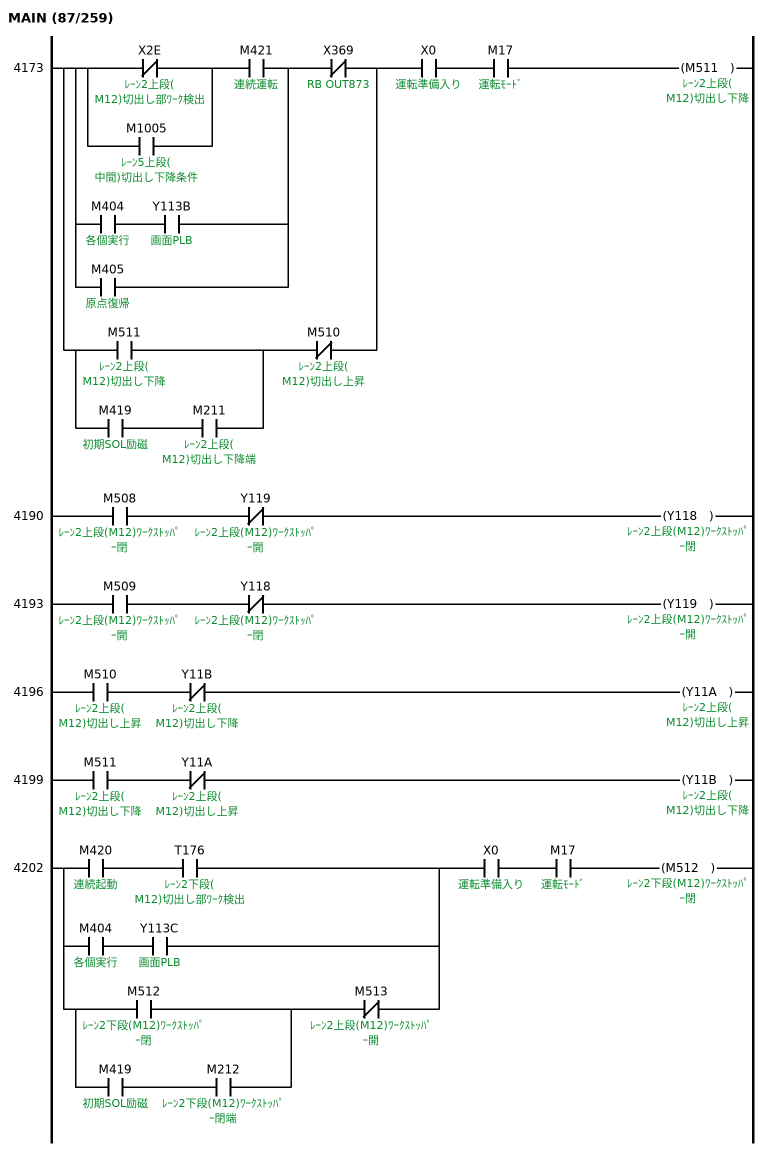
4173  LDI     X2E  ; ﾚｰﾝ2上段(M12)切出し部ﾜｰｸ検出
      OR      M1005  ; ﾚｰﾝ5上段(中間)切出し下降条件
      AND     M421  ; 連続運転
      LD      M404  ; 各個実行
      AND     Y113B  ; 画面PLB
      ORB
      OR      M405  ; 原点復帰
      ANI     X369  ; RB OUT873
      LD      M511  ; ﾚｰﾝ2上段(M12)切出し下降
      LD      M419  ; 初期SOL励磁
      AND     M211  ; ﾚｰﾝ2上段(M12)切出し下降端
      ORB
      ANI     M510  ; ﾚｰﾝ2上段(M12)切出し上昇
      ORB
      AND     X0  ; 運転準備入り
      AND     M17  ; 運転ﾓｰﾄﾞ
      OUT     M511  ; ﾚｰﾝ2上段(M12)切出し下降
4190  LD      M508  ; ﾚｰﾝ2上段(M12)ﾜｰｸｽﾄｯﾊﾟｰ閉
      ANI     Y119  ; ﾚｰﾝ2上段(M12)ﾜｰｸｽﾄｯﾊﾟｰ開
      OUT     Y118  ; ﾚｰﾝ2上段(M12)ﾜｰｸｽﾄｯﾊﾟｰ閉
4193  LD      M509  ; ﾚｰﾝ2上段(M12)ﾜｰｸｽﾄｯﾊﾟｰ開
      ANI     Y118  ; ﾚｰﾝ2上段(M12)ﾜｰｸｽﾄｯﾊﾟｰ閉
      OUT     Y119  ; ﾚｰﾝ2上段(M12)ﾜｰｸｽﾄｯﾊﾟｰ開
4196  LD      M510  ; ﾚｰﾝ2上段(M12)切出し上昇
      ANI     Y11B  ; ﾚｰﾝ2上段(M12)切出し下降
      OUT     Y11A  ; ﾚｰﾝ2上段(M12)切出し上昇
4199  LD      M511  ; ﾚｰﾝ2上段(M12)切出し下降
      ANI     Y11A  ; ﾚｰﾝ2上段(M12)切出し上昇
      OUT     Y11B  ; ﾚｰﾝ2上段(M12)切出し下降
4202  LD      M420  ; 連続起動
      AND     T176  ; ﾚｰﾝ2下段(M12)切出し部ﾜｰｸ検出
      LD      M404  ; 各個実行
      AND     Y113C  ; 画面PLB
      ORB
      LD      M512  ; ﾚｰﾝ2下段(M12)ﾜｰｸｽﾄｯﾊﾟｰ閉
      LD      M419  ; 初期SOL励磁
      AND     M212  ; ﾚｰﾝ2下段(M12)ﾜｰｸｽﾄｯﾊﾟｰ閉端
      ORB
      ANI     M513  ; ﾚｰﾝ2上段(M12)ﾜｰｸｽﾄｯﾊﾟｰ開
      ORB
      AND     X0  ; 運転準備入り
      AND     M17  ; 運転ﾓｰﾄﾞ
      OUT     M512  ; ﾚｰﾝ2下段(M12)ﾜｰｸｽﾄｯﾊﾟｰ閉
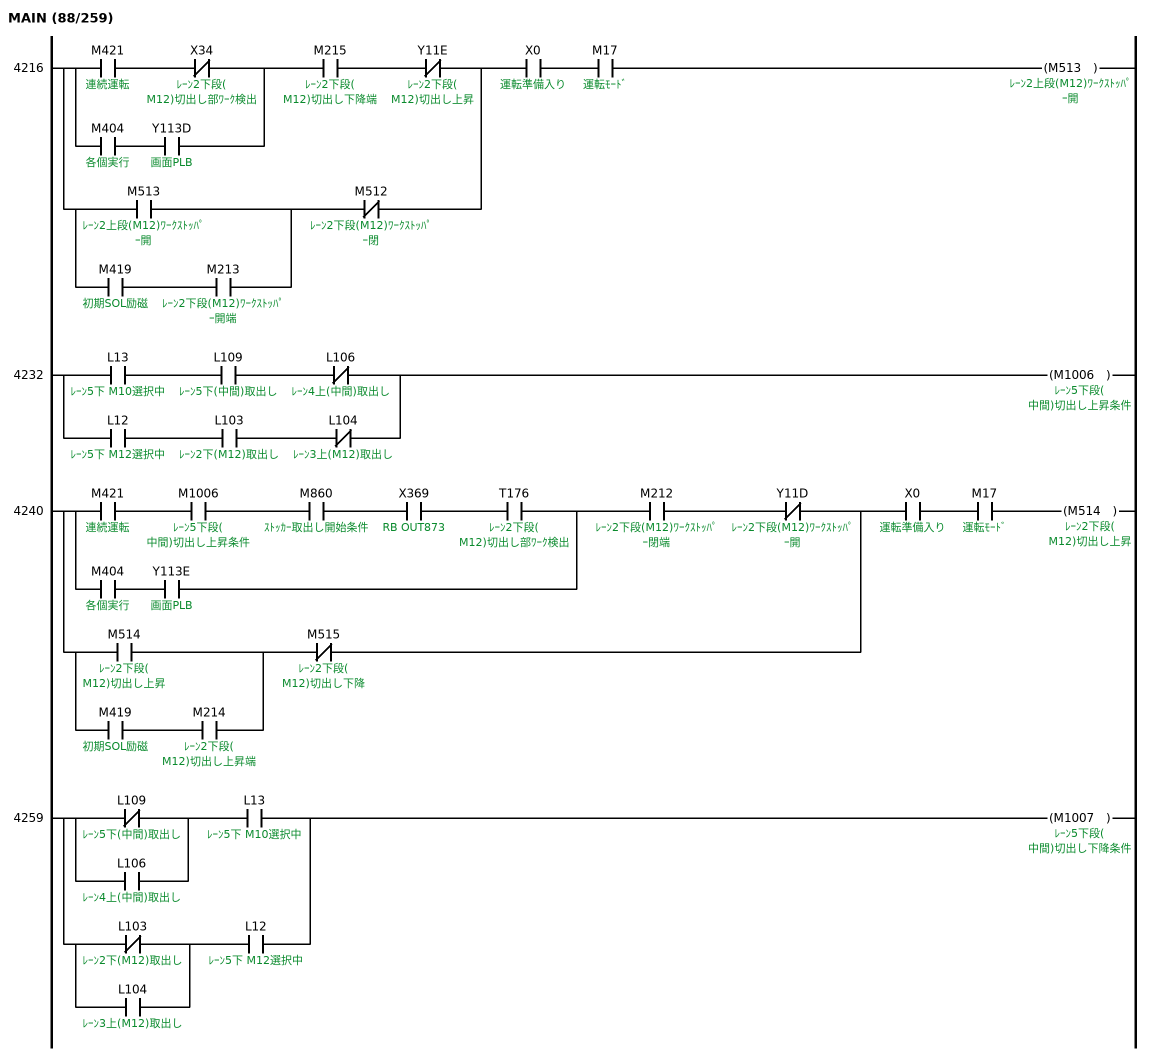
4216  LD      M421  ; 連続運転
      ANI     X34  ; ﾚｰﾝ2下段(M12)切出し部ﾜｰｸ検出
      LD      M404  ; 各個実行
      AND     Y113D  ; 画面PLB
      ORB
      AND     M215  ; ﾚｰﾝ2下段(M12)切出し下降端
      ANI     Y11E  ; ﾚｰﾝ2下段(M12)切出し上昇
      LD      M513  ; ﾚｰﾝ2上段(M12)ﾜｰｸｽﾄｯﾊﾟｰ開
      LD      M419  ; 初期SOL励磁
      AND     M213  ; ﾚｰﾝ2下段(M12)ﾜｰｸｽﾄｯﾊﾟｰ開端
      ORB
      ANI     M512  ; ﾚｰﾝ2下段(M12)ﾜｰｸｽﾄｯﾊﾟｰ閉
      ORB
      AND     X0  ; 運転準備入り
      AND     M17  ; 運転ﾓｰﾄﾞ
      OUT     M513  ; ﾚｰﾝ2上段(M12)ﾜｰｸｽﾄｯﾊﾟｰ開
4232  LD      L13  ; ﾚｰﾝ5下 M10選択中
      AND     L109  ; ﾚｰﾝ5下(中間)取出し
      ANI     L106  ; ﾚｰﾝ4上(中間)取出し
      LD      L12  ; ﾚｰﾝ5下 M12選択中
      AND     L103  ; ﾚｰﾝ2下(M12)取出し
      ANI     L104  ; ﾚｰﾝ3上(M12)取出し
      ORB
      OUT     M1006  ; ﾚｰﾝ5下段(中間)切出し上昇条件
4240  LD      M421  ; 連続運転
      AND     M1006  ; ﾚｰﾝ5下段(中間)切出し上昇条件
      AND     M860  ; ｽﾄｯｶｰ取出し開始条件
      AND     X369  ; RB OUT873
      AND     T176  ; ﾚｰﾝ2下段(M12)切出し部ﾜｰｸ検出
      LD      M404  ; 各個実行
      AND     Y113E  ; 画面PLB
      ORB
      AND     M212  ; ﾚｰﾝ2下段(M12)ﾜｰｸｽﾄｯﾊﾟｰ閉端
      ANI     Y11D  ; ﾚｰﾝ2下段(M12)ﾜｰｸｽﾄｯﾊﾟｰ開
      LD      M514  ; ﾚｰﾝ2下段(M12)切出し上昇
      LD      M419  ; 初期SOL励磁
      AND     M214  ; ﾚｰﾝ2下段(M12)切出し上昇端
      ORB
      ANI     M515  ; ﾚｰﾝ2下段(M12)切出し下降
      ORB
      AND     X0  ; 運転準備入り
      AND     M17  ; 運転ﾓｰﾄﾞ
      OUT     M514  ; ﾚｰﾝ2下段(M12)切出し上昇
4259  LDI     L109  ; ﾚｰﾝ5下(中間)取出し
      OR      L106  ; ﾚｰﾝ4上(中間)取出し
      AND     L13  ; ﾚｰﾝ5下 M10選択中
      LDI     L103  ; ﾚｰﾝ2下(M12)取出し
      OR      L104  ; ﾚｰﾝ3上(M12)取出し
      AND     L12  ; ﾚｰﾝ5下 M12選択中
      ORB
      OUT     M1007  ; ﾚｰﾝ5下段(中間)切出し下降条件
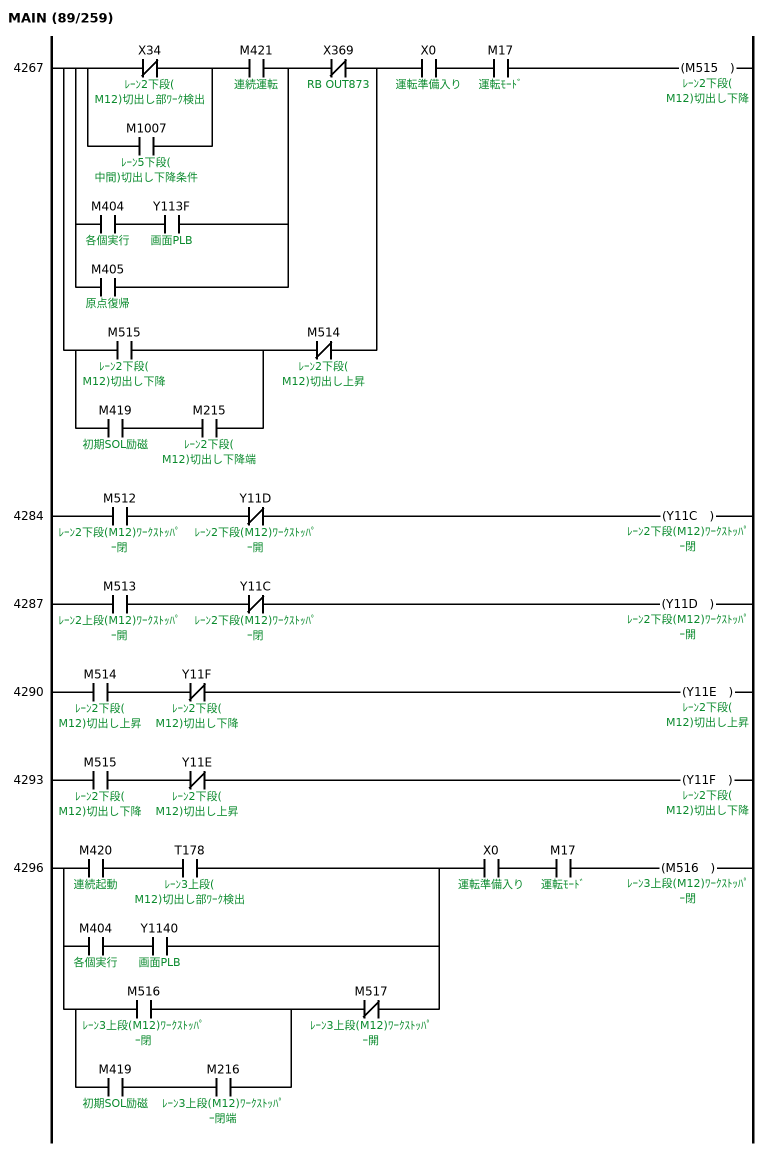
4267  LDI     X34  ; ﾚｰﾝ2下段(M12)切出し部ﾜｰｸ検出
      OR      M1007  ; ﾚｰﾝ5下段(中間)切出し下降条件
      AND     M421  ; 連続運転
      LD      M404  ; 各個実行
      AND     Y113F  ; 画面PLB
      ORB
      OR      M405  ; 原点復帰
      ANI     X369  ; RB OUT873
      LD      M515  ; ﾚｰﾝ2下段(M12)切出し下降
      LD      M419  ; 初期SOL励磁
      AND     M215  ; ﾚｰﾝ2下段(M12)切出し下降端
      ORB
      ANI     M514  ; ﾚｰﾝ2下段(M12)切出し上昇
      ORB
      AND     X0  ; 運転準備入り
      AND     M17  ; 運転ﾓｰﾄﾞ
      OUT     M515  ; ﾚｰﾝ2下段(M12)切出し下降
4284  LD      M512  ; ﾚｰﾝ2下段(M12)ﾜｰｸｽﾄｯﾊﾟｰ閉
      ANI     Y11D  ; ﾚｰﾝ2下段(M12)ﾜｰｸｽﾄｯﾊﾟｰ開
      OUT     Y11C  ; ﾚｰﾝ2下段(M12)ﾜｰｸｽﾄｯﾊﾟｰ閉
4287  LD      M513  ; ﾚｰﾝ2上段(M12)ﾜｰｸｽﾄｯﾊﾟｰ開
      ANI     Y11C  ; ﾚｰﾝ2下段(M12)ﾜｰｸｽﾄｯﾊﾟｰ閉
      OUT     Y11D  ; ﾚｰﾝ2下段(M12)ﾜｰｸｽﾄｯﾊﾟｰ開
4290  LD      M514  ; ﾚｰﾝ2下段(M12)切出し上昇
      ANI     Y11F  ; ﾚｰﾝ2下段(M12)切出し下降
      OUT     Y11E  ; ﾚｰﾝ2下段(M12)切出し上昇
4293  LD      M515  ; ﾚｰﾝ2下段(M12)切出し下降
      ANI     Y11E  ; ﾚｰﾝ2下段(M12)切出し上昇
      OUT     Y11F  ; ﾚｰﾝ2下段(M12)切出し下降
4296  LD      M420  ; 連続起動
      AND     T178  ; ﾚｰﾝ3上段(M12)切出し部ﾜｰｸ検出
      LD      M404  ; 各個実行
      AND     Y1140  ; 画面PLB
      ORB
      LD      M516  ; ﾚｰﾝ3上段(M12)ﾜｰｸｽﾄｯﾊﾟｰ閉
      LD      M419  ; 初期SOL励磁
      AND     M216  ; ﾚｰﾝ3上段(M12)ﾜｰｸｽﾄｯﾊﾟｰ閉端
      ORB
      ANI     M517  ; ﾚｰﾝ3上段(M12)ﾜｰｸｽﾄｯﾊﾟｰ開
      ORB
      AND     X0  ; 運転準備入り
      AND     M17  ; 運転ﾓｰﾄﾞ
      OUT     M516  ; ﾚｰﾝ3上段(M12)ﾜｰｸｽﾄｯﾊﾟｰ閉
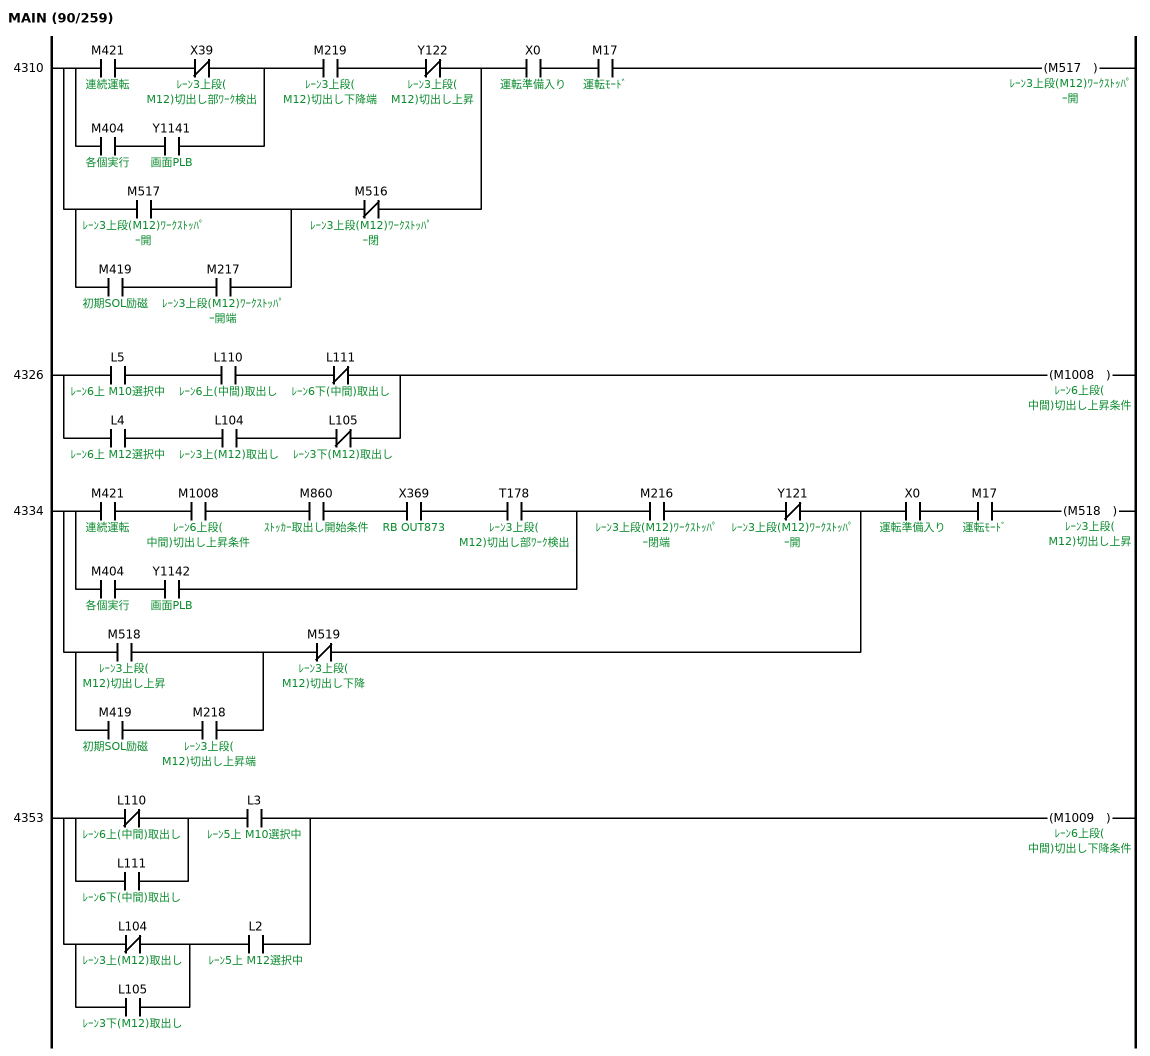
4310  LD      M421  ; 連続運転
      ANI     X39  ; ﾚｰﾝ3上段(M12)切出し部ﾜｰｸ検出
      LD      M404  ; 各個実行
      AND     Y1141  ; 画面PLB
      ORB
      AND     M219  ; ﾚｰﾝ3上段(M12)切出し下降端
      ANI     Y122  ; ﾚｰﾝ3上段(M12)切出し上昇
      LD      M517  ; ﾚｰﾝ3上段(M12)ﾜｰｸｽﾄｯﾊﾟｰ開
      LD      M419  ; 初期SOL励磁
      AND     M217  ; ﾚｰﾝ3上段(M12)ﾜｰｸｽﾄｯﾊﾟｰ開端
      ORB
      ANI     M516  ; ﾚｰﾝ3上段(M12)ﾜｰｸｽﾄｯﾊﾟｰ閉
      ORB
      AND     X0  ; 運転準備入り
      AND     M17  ; 運転ﾓｰﾄﾞ
      OUT     M517  ; ﾚｰﾝ3上段(M12)ﾜｰｸｽﾄｯﾊﾟｰ開
4326  LD      L5  ; ﾚｰﾝ6上 M10選択中
      AND     L110  ; ﾚｰﾝ6上(中間)取出し
      ANI     L111  ; ﾚｰﾝ6下(中間)取出し
      LD      L4  ; ﾚｰﾝ6上 M12選択中
      AND     L104  ; ﾚｰﾝ3上(M12)取出し
      ANI     L105  ; ﾚｰﾝ3下(M12)取出し
      ORB
      OUT     M1008  ; ﾚｰﾝ6上段(中間)切出し上昇条件
4334  LD      M421  ; 連続運転
      AND     M1008  ; ﾚｰﾝ6上段(中間)切出し上昇条件
      AND     M860  ; ｽﾄｯｶｰ取出し開始条件
      AND     X369  ; RB OUT873
      AND     T178  ; ﾚｰﾝ3上段(M12)切出し部ﾜｰｸ検出
      LD      M404  ; 各個実行
      AND     Y1142  ; 画面PLB
      ORB
      AND     M216  ; ﾚｰﾝ3上段(M12)ﾜｰｸｽﾄｯﾊﾟｰ閉端
      ANI     Y121  ; ﾚｰﾝ3上段(M12)ﾜｰｸｽﾄｯﾊﾟｰ開
      LD      M518  ; ﾚｰﾝ3上段(M12)切出し上昇
      LD      M419  ; 初期SOL励磁
      AND     M218  ; ﾚｰﾝ3上段(M12)切出し上昇端
      ORB
      ANI     M519  ; ﾚｰﾝ3上段(M12)切出し下降
      ORB
      AND     X0  ; 運転準備入り
      AND     M17  ; 運転ﾓｰﾄﾞ
      OUT     M518  ; ﾚｰﾝ3上段(M12)切出し上昇
4353  LDI     L110  ; ﾚｰﾝ6上(中間)取出し
      OR      L111  ; ﾚｰﾝ6下(中間)取出し
      AND     L3  ; ﾚｰﾝ5上 M10選択中
      LDI     L104  ; ﾚｰﾝ3上(M12)取出し
      OR      L105  ; ﾚｰﾝ3下(M12)取出し
      AND     L2  ; ﾚｰﾝ5上 M12選択中
      ORB
      OUT     M1009  ; ﾚｰﾝ6上段(中間)切出し下降条件
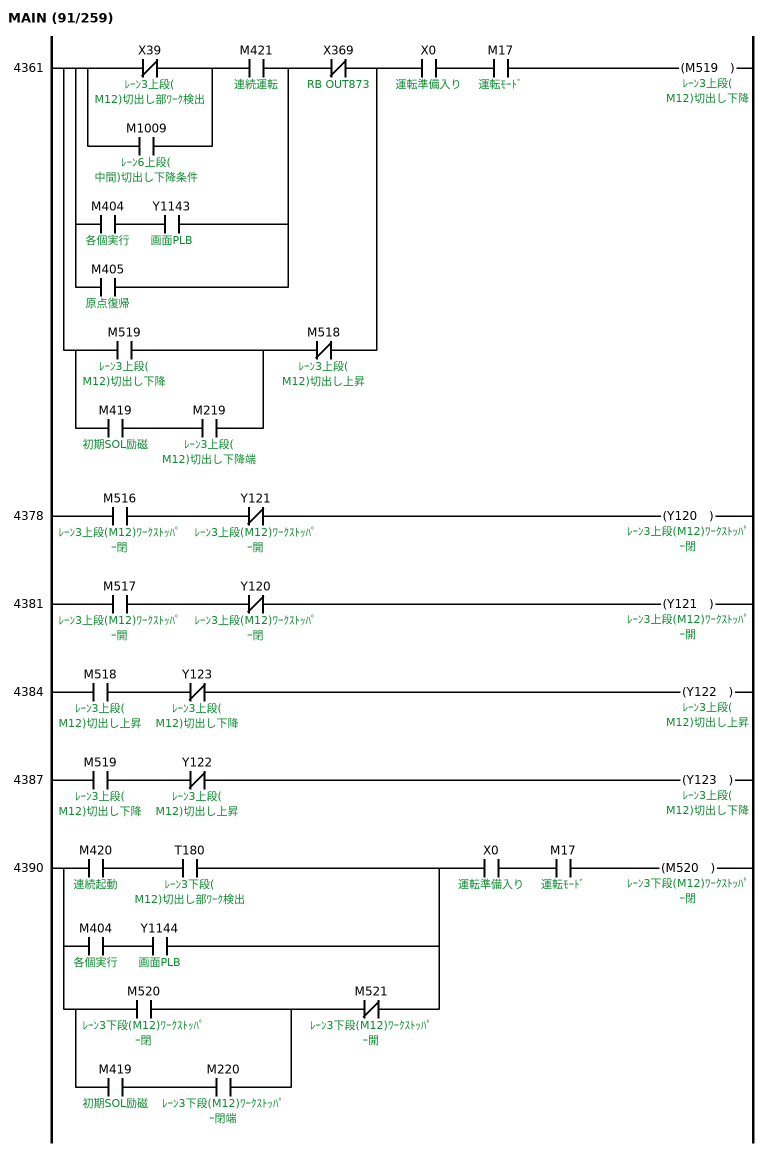
4361  LDI     X39  ; ﾚｰﾝ3上段(M12)切出し部ﾜｰｸ検出
      OR      M1009  ; ﾚｰﾝ6上段(中間)切出し下降条件
      AND     M421  ; 連続運転
      LD      M404  ; 各個実行
      AND     Y1143  ; 画面PLB
      ORB
      OR      M405  ; 原点復帰
      ANI     X369  ; RB OUT873
      LD      M519  ; ﾚｰﾝ3上段(M12)切出し下降
      LD      M419  ; 初期SOL励磁
      AND     M219  ; ﾚｰﾝ3上段(M12)切出し下降端
      ORB
      ANI     M518  ; ﾚｰﾝ3上段(M12)切出し上昇
      ORB
      AND     X0  ; 運転準備入り
      AND     M17  ; 運転ﾓｰﾄﾞ
      OUT     M519  ; ﾚｰﾝ3上段(M12)切出し下降
4378  LD      M516  ; ﾚｰﾝ3上段(M12)ﾜｰｸｽﾄｯﾊﾟｰ閉
      ANI     Y121  ; ﾚｰﾝ3上段(M12)ﾜｰｸｽﾄｯﾊﾟｰ開
      OUT     Y120  ; ﾚｰﾝ3上段(M12)ﾜｰｸｽﾄｯﾊﾟｰ閉
4381  LD      M517  ; ﾚｰﾝ3上段(M12)ﾜｰｸｽﾄｯﾊﾟｰ開
      ANI     Y120  ; ﾚｰﾝ3上段(M12)ﾜｰｸｽﾄｯﾊﾟｰ閉
      OUT     Y121  ; ﾚｰﾝ3上段(M12)ﾜｰｸｽﾄｯﾊﾟｰ開
4384  LD      M518  ; ﾚｰﾝ3上段(M12)切出し上昇
      ANI     Y123  ; ﾚｰﾝ3上段(M12)切出し下降
      OUT     Y122  ; ﾚｰﾝ3上段(M12)切出し上昇
4387  LD      M519  ; ﾚｰﾝ3上段(M12)切出し下降
      ANI     Y122  ; ﾚｰﾝ3上段(M12)切出し上昇
      OUT     Y123  ; ﾚｰﾝ3上段(M12)切出し下降
4390  LD      M420  ; 連続起動
      AND     T180  ; ﾚｰﾝ3下段(M12)切出し部ﾜｰｸ検出
      LD      M404  ; 各個実行
      AND     Y1144  ; 画面PLB
      ORB
      LD      M520  ; ﾚｰﾝ3下段(M12)ﾜｰｸｽﾄｯﾊﾟｰ閉
      LD      M419  ; 初期SOL励磁
      AND     M220  ; ﾚｰﾝ3下段(M12)ﾜｰｸｽﾄｯﾊﾟｰ閉端
      ORB
      ANI     M521  ; ﾚｰﾝ3下段(M12)ﾜｰｸｽﾄｯﾊﾟｰ開
      ORB
      AND     X0  ; 運転準備入り
      AND     M17  ; 運転ﾓｰﾄﾞ
      OUT     M520  ; ﾚｰﾝ3下段(M12)ﾜｰｸｽﾄｯﾊﾟｰ閉
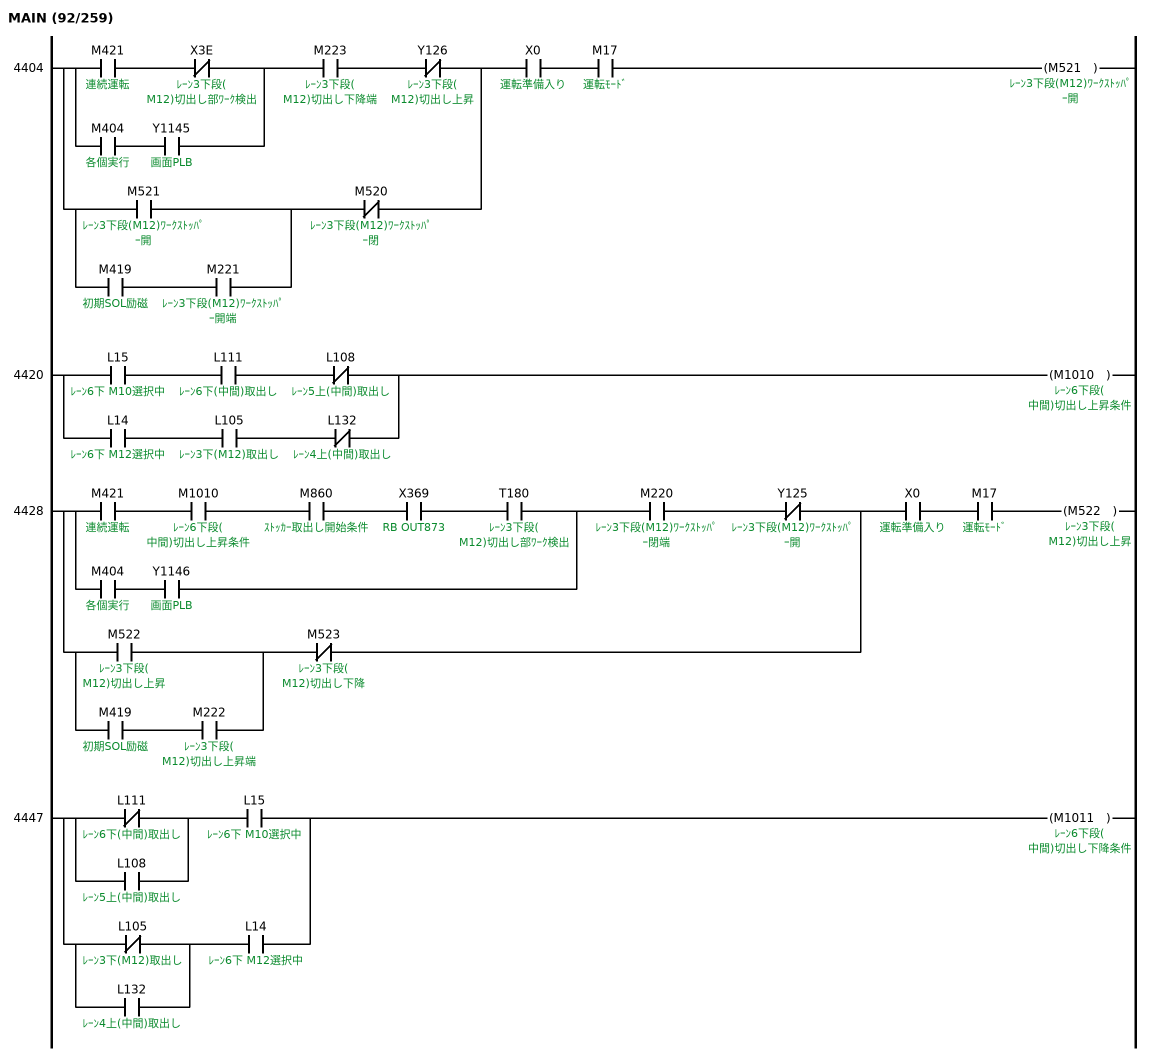
4404  LD      M421  ; 連続運転
      ANI     X3E  ; ﾚｰﾝ3下段(M12)切出し部ﾜｰｸ検出
      LD      M404  ; 各個実行
      AND     Y1145  ; 画面PLB
      ORB
      AND     M223  ; ﾚｰﾝ3下段(M12)切出し下降端
      ANI     Y126  ; ﾚｰﾝ3下段(M12)切出し上昇
      LD      M521  ; ﾚｰﾝ3下段(M12)ﾜｰｸｽﾄｯﾊﾟｰ開
      LD      M419  ; 初期SOL励磁
      AND     M221  ; ﾚｰﾝ3下段(M12)ﾜｰｸｽﾄｯﾊﾟｰ開端
      ORB
      ANI     M520  ; ﾚｰﾝ3下段(M12)ﾜｰｸｽﾄｯﾊﾟｰ閉
      ORB
      AND     X0  ; 運転準備入り
      AND     M17  ; 運転ﾓｰﾄﾞ
      OUT     M521  ; ﾚｰﾝ3下段(M12)ﾜｰｸｽﾄｯﾊﾟｰ開
4420  LD      L15  ; ﾚｰﾝ6下 M10選択中
      AND     L111  ; ﾚｰﾝ6下(中間)取出し
      ANI     L108  ; ﾚｰﾝ5上(中間)取出し
      LD      L14  ; ﾚｰﾝ6下 M12選択中
      AND     L105  ; ﾚｰﾝ3下(M12)取出し
      ANI     L132  ; ﾚｰﾝ4上(中間)取出し
      ORB
      OUT     M1010  ; ﾚｰﾝ6下段(中間)切出し上昇条件
4428  LD      M421  ; 連続運転
      AND     M1010  ; ﾚｰﾝ6下段(中間)切出し上昇条件
      AND     M860  ; ｽﾄｯｶｰ取出し開始条件
      AND     X369  ; RB OUT873
      AND     T180  ; ﾚｰﾝ3下段(M12)切出し部ﾜｰｸ検出
      LD      M404  ; 各個実行
      AND     Y1146  ; 画面PLB
      ORB
      AND     M220  ; ﾚｰﾝ3下段(M12)ﾜｰｸｽﾄｯﾊﾟｰ閉端
      ANI     Y125  ; ﾚｰﾝ3下段(M12)ﾜｰｸｽﾄｯﾊﾟｰ開
      LD      M522  ; ﾚｰﾝ3下段(M12)切出し上昇
      LD      M419  ; 初期SOL励磁
      AND     M222  ; ﾚｰﾝ3下段(M12)切出し上昇端
      ORB
      ANI     M523  ; ﾚｰﾝ3下段(M12)切出し下降
      ORB
      AND     X0  ; 運転準備入り
      AND     M17  ; 運転ﾓｰﾄﾞ
      OUT     M522  ; ﾚｰﾝ3下段(M12)切出し上昇
4447  LDI     L111  ; ﾚｰﾝ6下(中間)取出し
      OR      L108  ; ﾚｰﾝ5上(中間)取出し
      AND     L15  ; ﾚｰﾝ6下 M10選択中
      LDI     L105  ; ﾚｰﾝ3下(M12)取出し
      OR      L132  ; ﾚｰﾝ4上(中間)取出し
      AND     L14  ; ﾚｰﾝ6下 M12選択中
      ORB
      OUT     M1011  ; ﾚｰﾝ6下段(中間)切出し下降条件
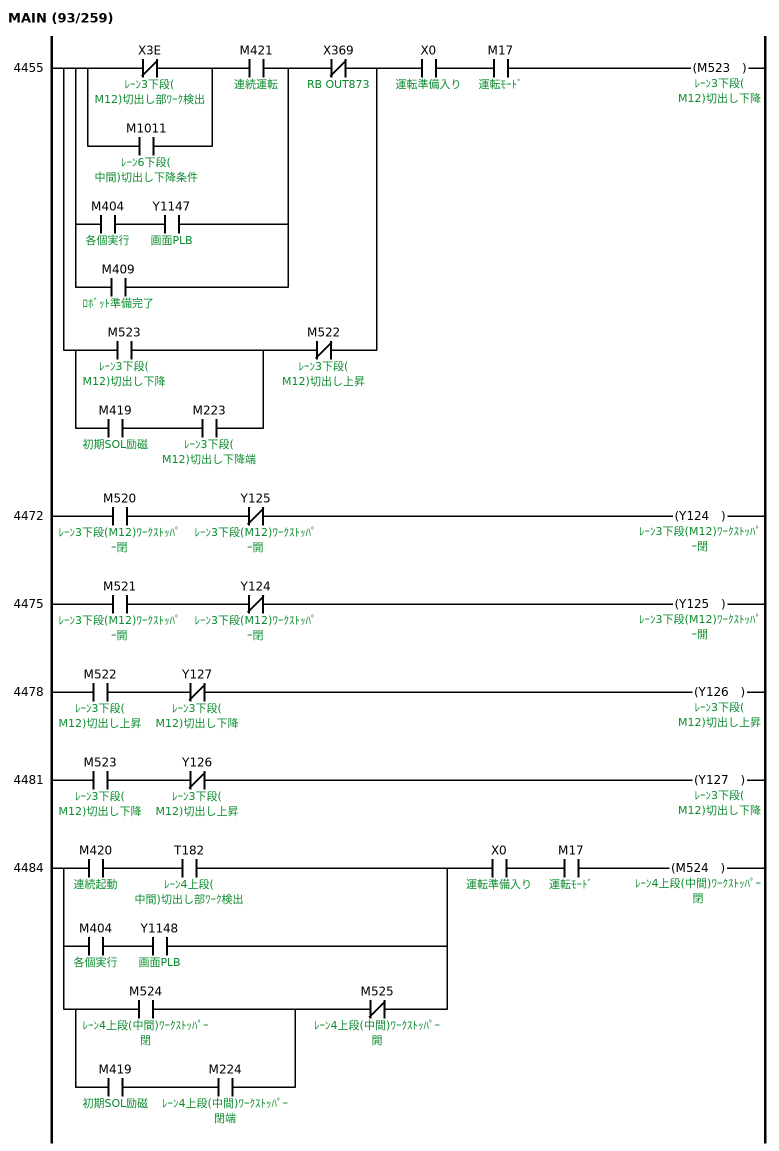
4455  LDI     X3E  ; ﾚｰﾝ3下段(M12)切出し部ﾜｰｸ検出
      OR      M1011  ; ﾚｰﾝ6下段(中間)切出し下降条件
      AND     M421  ; 連続運転
      LD      M404  ; 各個実行
      AND     Y1147  ; 画面PLB
      ORB
      OR      M409  ; ﾛﾎﾞｯﾄ準備完了
      ANI     X369  ; RB OUT873
      LD      M523  ; ﾚｰﾝ3下段(M12)切出し下降
      LD      M419  ; 初期SOL励磁
      AND     M223  ; ﾚｰﾝ3下段(M12)切出し下降端
      ORB
      ANI     M522  ; ﾚｰﾝ3下段(M12)切出し上昇
      ORB
      AND     X0  ; 運転準備入り
      AND     M17  ; 運転ﾓｰﾄﾞ
      OUT     M523  ; ﾚｰﾝ3下段(M12)切出し下降
4472  LD      M520  ; ﾚｰﾝ3下段(M12)ﾜｰｸｽﾄｯﾊﾟｰ閉
      ANI     Y125  ; ﾚｰﾝ3下段(M12)ﾜｰｸｽﾄｯﾊﾟｰ開
      OUT     Y124  ; ﾚｰﾝ3下段(M12)ﾜｰｸｽﾄｯﾊﾟｰ閉
4475  LD      M521  ; ﾚｰﾝ3下段(M12)ﾜｰｸｽﾄｯﾊﾟｰ開
      ANI     Y124  ; ﾚｰﾝ3下段(M12)ﾜｰｸｽﾄｯﾊﾟｰ閉
      OUT     Y125  ; ﾚｰﾝ3下段(M12)ﾜｰｸｽﾄｯﾊﾟｰ開
4478  LD      M522  ; ﾚｰﾝ3下段(M12)切出し上昇
      ANI     Y127  ; ﾚｰﾝ3下段(M12)切出し下降
      OUT     Y126  ; ﾚｰﾝ3下段(M12)切出し上昇
4481  LD      M523  ; ﾚｰﾝ3下段(M12)切出し下降
      ANI     Y126  ; ﾚｰﾝ3下段(M12)切出し上昇
      OUT     Y127  ; ﾚｰﾝ3下段(M12)切出し下降
4484  LD      M420  ; 連続起動
      AND     T182  ; ﾚｰﾝ4上段(中間)切出し部ﾜｰｸ検出
      LD      M404  ; 各個実行
      AND     Y1148  ; 画面PLB
      ORB
      LD      M524  ; ﾚｰﾝ4上段(中間)ﾜｰｸｽﾄｯﾊﾟｰ閉
      LD      M419  ; 初期SOL励磁
      AND     M224  ; ﾚｰﾝ4上段(中間)ﾜｰｸｽﾄｯﾊﾟｰ閉端
      ORB
      ANI     M525  ; ﾚｰﾝ4上段(中間)ﾜｰｸｽﾄｯﾊﾟｰ開
      ORB
      AND     X0  ; 運転準備入り
      AND     M17  ; 運転ﾓｰﾄﾞ
      OUT     M524  ; ﾚｰﾝ4上段(中間)ﾜｰｸｽﾄｯﾊﾟｰ閉
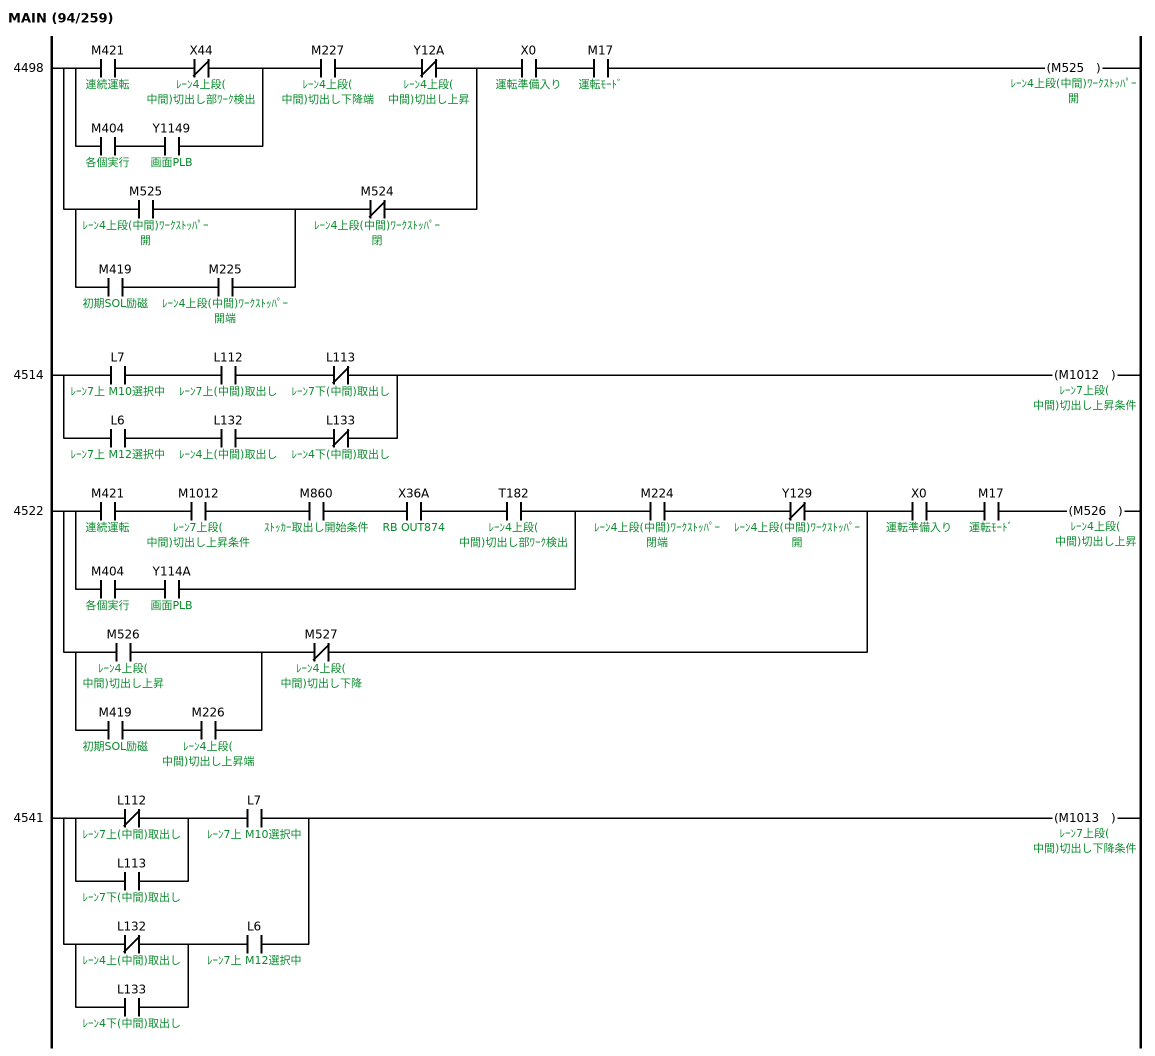
4498  LD      M421  ; 連続運転
      ANI     X44  ; ﾚｰﾝ4上段(中間)切出し部ﾜｰｸ検出
      LD      M404  ; 各個実行
      AND     Y1149  ; 画面PLB
      ORB
      AND     M227  ; ﾚｰﾝ4上段(中間)切出し下降端
      ANI     Y12A  ; ﾚｰﾝ4上段(中間)切出し上昇
      LD      M525  ; ﾚｰﾝ4上段(中間)ﾜｰｸｽﾄｯﾊﾟｰ開
      LD      M419  ; 初期SOL励磁
      AND     M225  ; ﾚｰﾝ4上段(中間)ﾜｰｸｽﾄｯﾊﾟｰ開端
      ORB
      ANI     M524  ; ﾚｰﾝ4上段(中間)ﾜｰｸｽﾄｯﾊﾟｰ閉
      ORB
      AND     X0  ; 運転準備入り
      AND     M17  ; 運転ﾓｰﾄﾞ
      OUT     M525  ; ﾚｰﾝ4上段(中間)ﾜｰｸｽﾄｯﾊﾟｰ開
4514  LD      L7  ; ﾚｰﾝ7上 M10選択中
      AND     L112  ; ﾚｰﾝ7上(中間)取出し
      ANI     L113  ; ﾚｰﾝ7下(中間)取出し
      LD      L6  ; ﾚｰﾝ7上 M12選択中
      AND     L132  ; ﾚｰﾝ4上(中間)取出し
      ANI     L133  ; ﾚｰﾝ4下(中間)取出し
      ORB
      OUT     M1012  ; ﾚｰﾝ7上段(中間)切出し上昇条件
4522  LD      M421  ; 連続運転
      AND     M1012  ; ﾚｰﾝ7上段(中間)切出し上昇条件
      AND     M860  ; ｽﾄｯｶｰ取出し開始条件
      AND     X36A  ; RB OUT874
      AND     T182  ; ﾚｰﾝ4上段(中間)切出し部ﾜｰｸ検出
      LD      M404  ; 各個実行
      AND     Y114A  ; 画面PLB
      ORB
      AND     M224  ; ﾚｰﾝ4上段(中間)ﾜｰｸｽﾄｯﾊﾟｰ閉端
      ANI     Y129  ; ﾚｰﾝ4上段(中間)ﾜｰｸｽﾄｯﾊﾟｰ開
      LD      M526  ; ﾚｰﾝ4上段(中間)切出し上昇
      LD      M419  ; 初期SOL励磁
      AND     M226  ; ﾚｰﾝ4上段(中間)切出し上昇端
      ORB
      ANI     M527  ; ﾚｰﾝ4上段(中間)切出し下降
      ORB
      AND     X0  ; 運転準備入り
      AND     M17  ; 運転ﾓｰﾄﾞ
      OUT     M526  ; ﾚｰﾝ4上段(中間)切出し上昇
4541  LDI     L112  ; ﾚｰﾝ7上(中間)取出し
      OR      L113  ; ﾚｰﾝ7下(中間)取出し
      AND     L7  ; ﾚｰﾝ7上 M10選択中
      LDI     L132  ; ﾚｰﾝ4上(中間)取出し
      OR      L133  ; ﾚｰﾝ4下(中間)取出し
      AND     L6  ; ﾚｰﾝ7上 M12選択中
      ORB
      OUT     M1013  ; ﾚｰﾝ7上段(中間)切出し下降条件
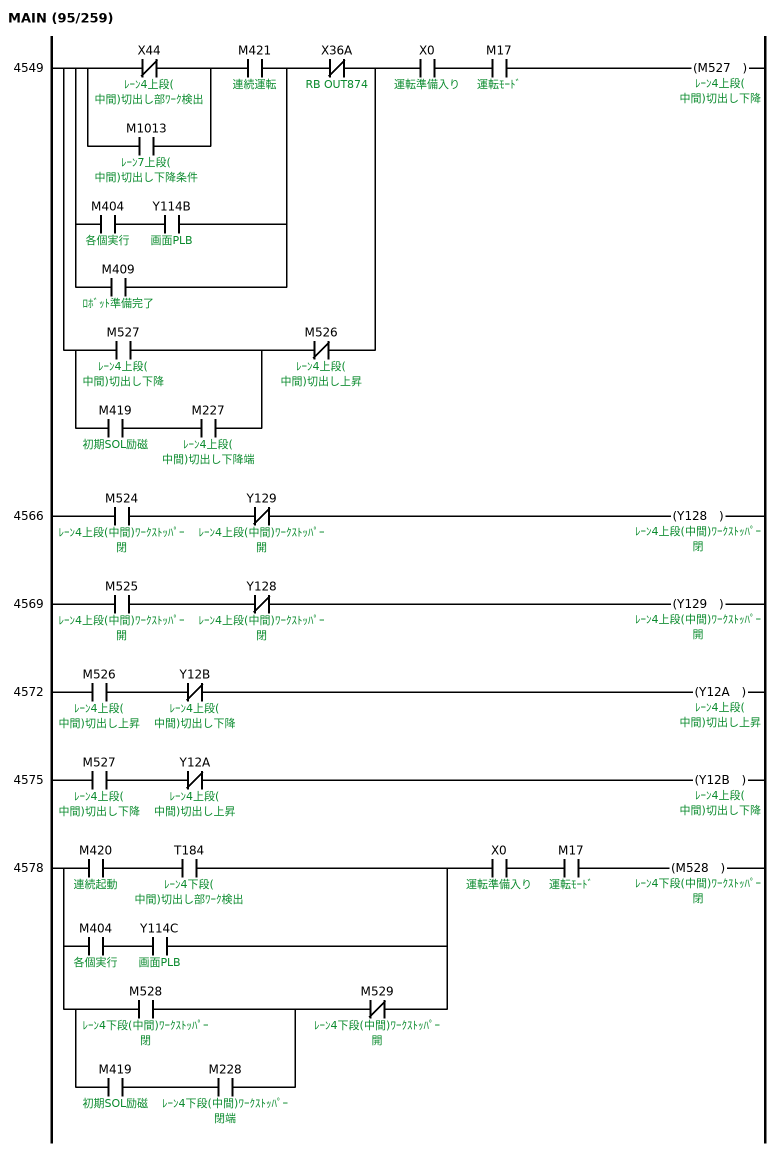
4549  LDI     X44  ; ﾚｰﾝ4上段(中間)切出し部ﾜｰｸ検出
      OR      M1013  ; ﾚｰﾝ7上段(中間)切出し下降条件
      AND     M421  ; 連続運転
      LD      M404  ; 各個実行
      AND     Y114B  ; 画面PLB
      ORB
      OR      M409  ; ﾛﾎﾞｯﾄ準備完了
      ANI     X36A  ; RB OUT874
      LD      M527  ; ﾚｰﾝ4上段(中間)切出し下降
      LD      M419  ; 初期SOL励磁
      AND     M227  ; ﾚｰﾝ4上段(中間)切出し下降端
      ORB
      ANI     M526  ; ﾚｰﾝ4上段(中間)切出し上昇
      ORB
      AND     X0  ; 運転準備入り
      AND     M17  ; 運転ﾓｰﾄﾞ
      OUT     M527  ; ﾚｰﾝ4上段(中間)切出し下降
4566  LD      M524  ; ﾚｰﾝ4上段(中間)ﾜｰｸｽﾄｯﾊﾟｰ閉
      ANI     Y129  ; ﾚｰﾝ4上段(中間)ﾜｰｸｽﾄｯﾊﾟｰ開
      OUT     Y128  ; ﾚｰﾝ4上段(中間)ﾜｰｸｽﾄｯﾊﾟｰ閉
4569  LD      M525  ; ﾚｰﾝ4上段(中間)ﾜｰｸｽﾄｯﾊﾟｰ開
      ANI     Y128  ; ﾚｰﾝ4上段(中間)ﾜｰｸｽﾄｯﾊﾟｰ閉
      OUT     Y129  ; ﾚｰﾝ4上段(中間)ﾜｰｸｽﾄｯﾊﾟｰ開
4572  LD      M526  ; ﾚｰﾝ4上段(中間)切出し上昇
      ANI     Y12B  ; ﾚｰﾝ4上段(中間)切出し下降
      OUT     Y12A  ; ﾚｰﾝ4上段(中間)切出し上昇
4575  LD      M527  ; ﾚｰﾝ4上段(中間)切出し下降
      ANI     Y12A  ; ﾚｰﾝ4上段(中間)切出し上昇
      OUT     Y12B  ; ﾚｰﾝ4上段(中間)切出し下降
4578  LD      M420  ; 連続起動
      AND     T184  ; ﾚｰﾝ4下段(中間)切出し部ﾜｰｸ検出
      LD      M404  ; 各個実行
      AND     Y114C  ; 画面PLB
      ORB
      LD      M528  ; ﾚｰﾝ4下段(中間)ﾜｰｸｽﾄｯﾊﾟｰ閉
      LD      M419  ; 初期SOL励磁
      AND     M228  ; ﾚｰﾝ4下段(中間)ﾜｰｸｽﾄｯﾊﾟｰ閉端
      ORB
      ANI     M529  ; ﾚｰﾝ4下段(中間)ﾜｰｸｽﾄｯﾊﾟｰ開
      ORB
      AND     X0  ; 運転準備入り
      AND     M17  ; 運転ﾓｰﾄﾞ
      OUT     M528  ; ﾚｰﾝ4下段(中間)ﾜｰｸｽﾄｯﾊﾟｰ閉
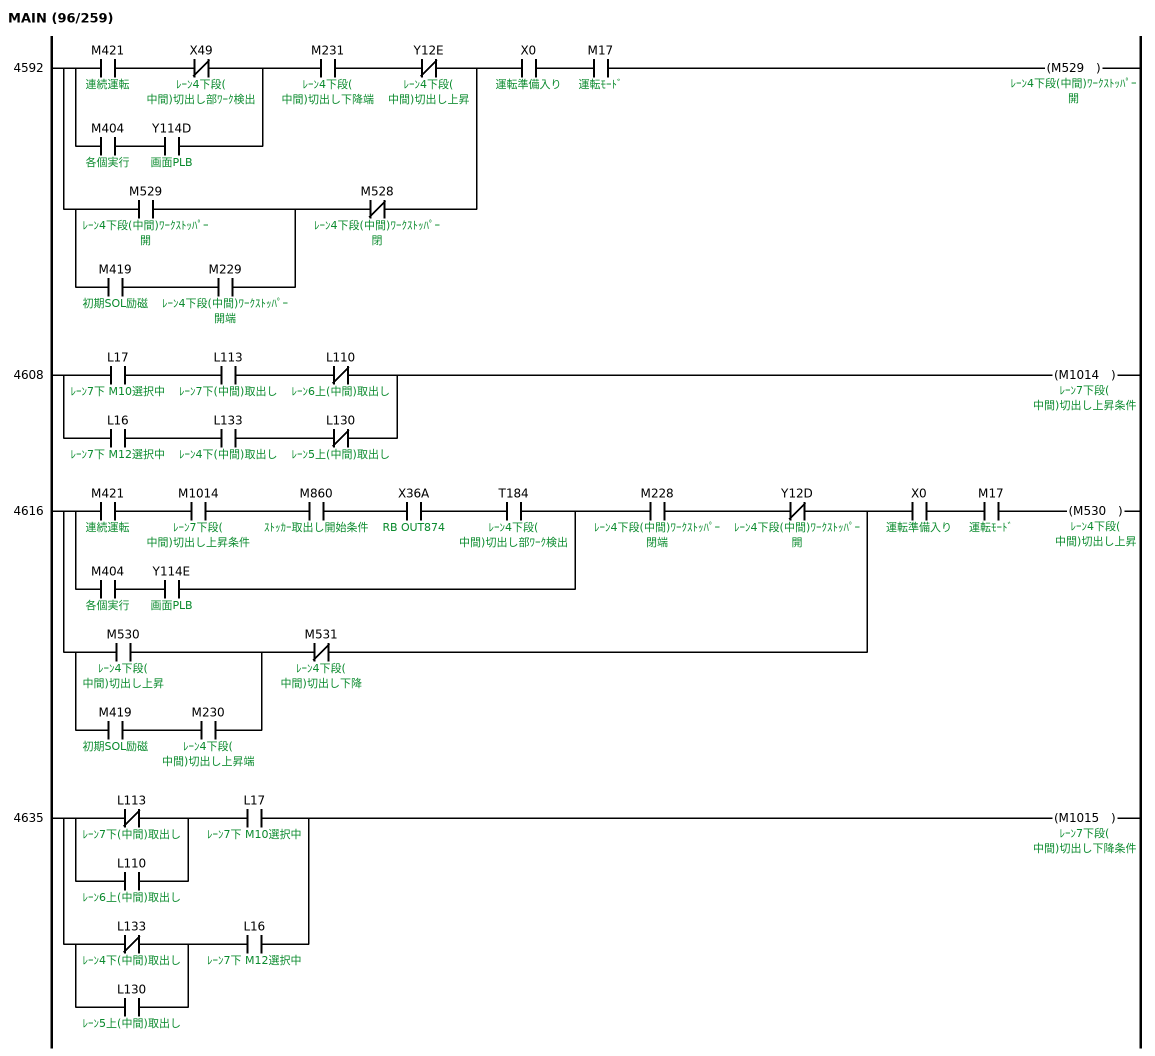
4592  LD      M421  ; 連続運転
      ANI     X49  ; ﾚｰﾝ4下段(中間)切出し部ﾜｰｸ検出
      LD      M404  ; 各個実行
      AND     Y114D  ; 画面PLB
      ORB
      AND     M231  ; ﾚｰﾝ4下段(中間)切出し下降端
      ANI     Y12E  ; ﾚｰﾝ4下段(中間)切出し上昇
      LD      M529  ; ﾚｰﾝ4下段(中間)ﾜｰｸｽﾄｯﾊﾟｰ開
      LD      M419  ; 初期SOL励磁
      AND     M229  ; ﾚｰﾝ4下段(中間)ﾜｰｸｽﾄｯﾊﾟｰ開端
      ORB
      ANI     M528  ; ﾚｰﾝ4下段(中間)ﾜｰｸｽﾄｯﾊﾟｰ閉
      ORB
      AND     X0  ; 運転準備入り
      AND     M17  ; 運転ﾓｰﾄﾞ
      OUT     M529  ; ﾚｰﾝ4下段(中間)ﾜｰｸｽﾄｯﾊﾟｰ開
4608  LD      L17  ; ﾚｰﾝ7下 M10選択中
      AND     L113  ; ﾚｰﾝ7下(中間)取出し
      ANI     L110  ; ﾚｰﾝ6上(中間)取出し
      LD      L16  ; ﾚｰﾝ7下 M12選択中
      AND     L133  ; ﾚｰﾝ4下(中間)取出し
      ANI     L130  ; ﾚｰﾝ5上(中間)取出し
      ORB
      OUT     M1014  ; ﾚｰﾝ7下段(中間)切出し上昇条件
4616  LD      M421  ; 連続運転
      AND     M1014  ; ﾚｰﾝ7下段(中間)切出し上昇条件
      AND     M860  ; ｽﾄｯｶｰ取出し開始条件
      AND     X36A  ; RB OUT874
      AND     T184  ; ﾚｰﾝ4下段(中間)切出し部ﾜｰｸ検出
      LD      M404  ; 各個実行
      AND     Y114E  ; 画面PLB
      ORB
      AND     M228  ; ﾚｰﾝ4下段(中間)ﾜｰｸｽﾄｯﾊﾟｰ閉端
      ANI     Y12D  ; ﾚｰﾝ4下段(中間)ﾜｰｸｽﾄｯﾊﾟｰ開
      LD      M530  ; ﾚｰﾝ4下段(中間)切出し上昇
      LD      M419  ; 初期SOL励磁
      AND     M230  ; ﾚｰﾝ4下段(中間)切出し上昇端
      ORB
      ANI     M531  ; ﾚｰﾝ4下段(中間)切出し下降
      ORB
      AND     X0  ; 運転準備入り
      AND     M17  ; 運転ﾓｰﾄﾞ
      OUT     M530  ; ﾚｰﾝ4下段(中間)切出し上昇
4635  LDI     L113  ; ﾚｰﾝ7下(中間)取出し
      OR      L110  ; ﾚｰﾝ6上(中間)取出し
      AND     L17  ; ﾚｰﾝ7下 M10選択中
      LDI     L133  ; ﾚｰﾝ4下(中間)取出し
      OR      L130  ; ﾚｰﾝ5上(中間)取出し
      AND     L16  ; ﾚｰﾝ7下 M12選択中
      ORB
      OUT     M1015  ; ﾚｰﾝ7下段(中間)切出し下降条件
